// Mitsubishi GX Works2 project: GDF-UV-4GC-20210804 souce   PLC: Q00U

PROGRAM MAIN
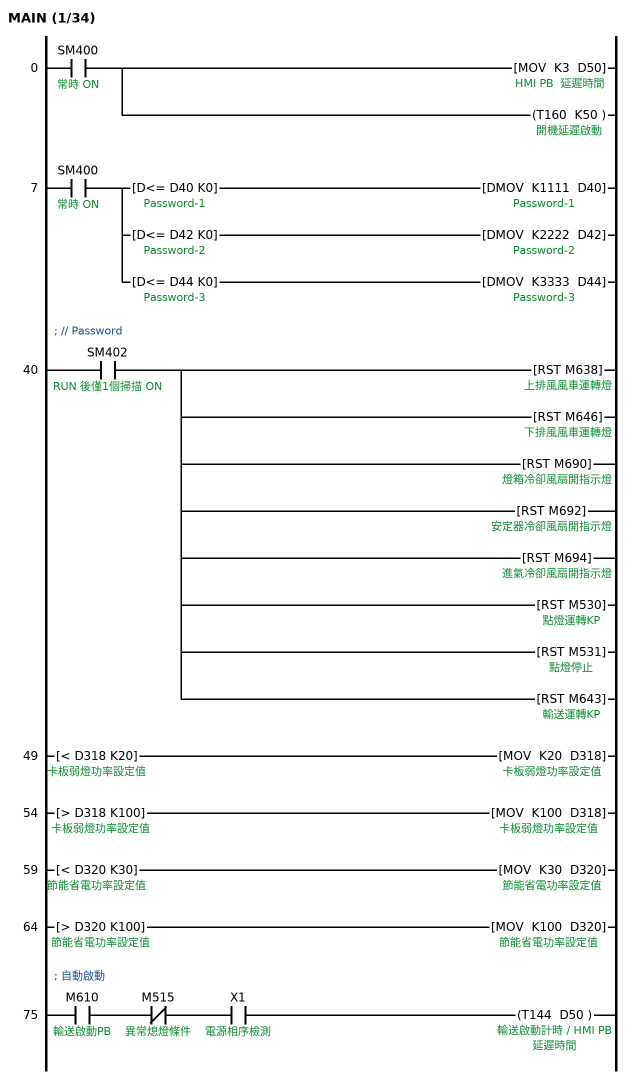
0     LD      SM400  ; 常時 ON
      MOV     K3 D50  ; HMI PB  延遲時間
      OUT     T160 K50  ; 開機延遲啟動
7     LD      SM400  ; 常時 ON
      MPS
      ANDD<=  D40 K0  ; Password-1
      DMOV    K1111 D40
      MRD
      ANDD<=  D42 K0  ; Password-2
      DMOV    K2222 D42
      MPP
      ANDD<=  D44 K0  ; Password-3
      DMOV    K3333 D44
; // Password
40    LD      SM402  ; RUN 後僅1個掃描 ON
      RST     M638  ; 上排風風車運轉燈
      RST     M646  ; 下排風風車運轉燈
      RST     M690  ; 燈箱冷卻風扇開指示燈
      RST     M692  ; 安定器冷卻風扇開指示燈
      RST     M694  ; 進氣冷卻風扇開指示燈
      RST     M530  ; 點燈運轉KP
      RST     M531  ; 點燈停止
      RST     M643  ; 輸送運轉KP
49    LD<     D318 K20  ; 卡板弱燈功率設定值
      MOV     K20 D318
54    LD>     D318 K100  ; 卡板弱燈功率設定值
      MOV     K100 D318
59    LD<     D320 K30  ; 節能省電功率設定值
      MOV     K30 D320
64    LD>     D320 K100  ; 節能省電功率設定值
      MOV     K100 D320
; 自動啟動
75    LD      M610  ; 輸送啟動PB
      ANI     M515  ; 異常熄燈條件
      AND     X1  ; 電源相序檢測
      OUT     T144 D50  ; 輸送啟動計時 / HMI PB  延遲時間
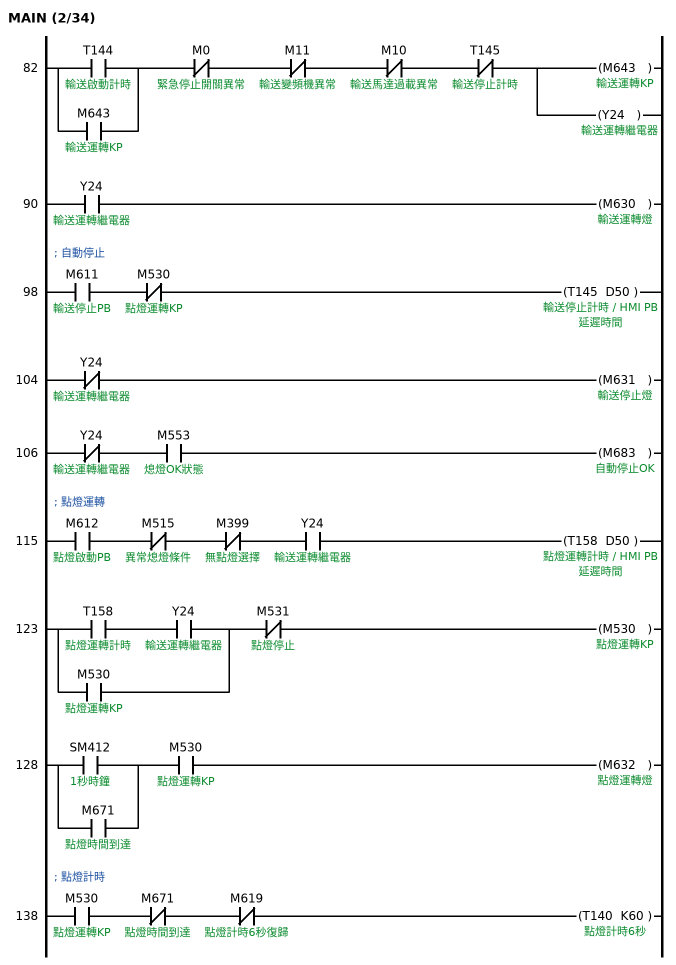
82    LD      T144  ; 輸送啟動計時
      OR      M643  ; 輸送運轉KP
      ANI     M0  ; 緊急停止開關異常
      ANI     M11  ; 輸送變頻機異常
      ANI     M10  ; 輸送馬達過載異常
      ANI     T145  ; 輸送停止計時
      OUT     M643  ; 輸送運轉KP
      OUT     Y24  ; 輸送運轉繼電器
90    LD      Y24  ; 輸送運轉繼電器
      OUT     M630  ; 輸送運轉燈
; 自動停止
98    LD      M611  ; 輸送停止PB
      ANI     M530  ; 點燈運轉KP
      OUT     T145 D50  ; 輸送停止計時 / HMI PB  延遲時間
104   LDI     Y24  ; 輸送運轉繼電器
      OUT     M631  ; 輸送停止燈
106   LDI     Y24  ; 輸送運轉繼電器
      AND     M553  ; 熄燈OK狀態
      OUT     M683  ; 自動停止OK
; 點燈運轉
115   LD      M612  ; 點燈啟動PB
      ANI     M515  ; 異常熄燈條件
      ANI     M399  ; 無點燈選擇
      AND     Y24  ; 輸送運轉繼電器
      OUT     T158 D50  ; 點燈運轉計時 / HMI PB  延遲時間
123   LD      T158  ; 點燈運轉計時
      AND     Y24  ; 輸送運轉繼電器
      OR      M530  ; 點燈運轉KP
      ANI     M531  ; 點燈停止
      OUT     M530  ; 點燈運轉KP
128   LD      SM412  ; 1秒時鐘
      OR      M671  ; 點燈時間到達
      AND     M530  ; 點燈運轉KP
      OUT     M632  ; 點燈運轉燈
; 點燈計時
138   LD      M530  ; 點燈運轉KP
      ANI     M671  ; 點燈時間到達
      ANI     M619  ; 點燈計時6秒復歸
      OUT     T140 K60  ; 點燈計時6秒
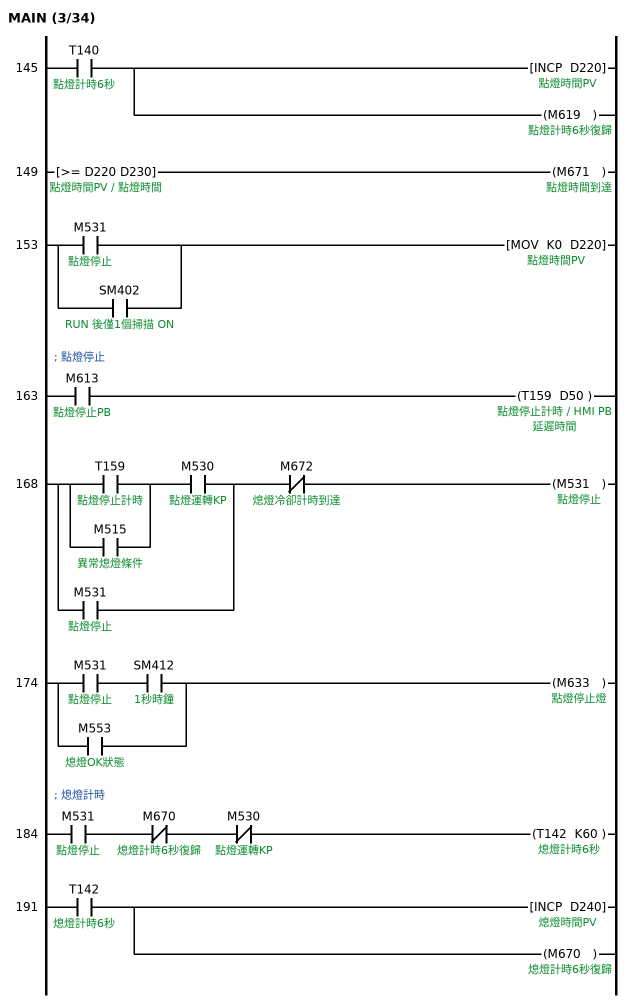
145   LD      T140  ; 點燈計時6秒
      INCP    D220  ; 點燈時間PV
      OUT     M619  ; 點燈計時6秒復歸
149   LD>=    D220 D230  ; 點燈時間PV / 點燈時間
      OUT     M671  ; 點燈時間到達
153   LD      M531  ; 點燈停止
      OR      SM402  ; RUN 後僅1個掃描 ON
      MOV     K0 D220
; 點燈停止
163   LD      M613  ; 點燈停止PB
      OUT     T159 D50  ; 點燈停止計時 / HMI PB  延遲時間
168   LD      T159  ; 點燈停止計時
      OR      M515  ; 異常熄燈條件
      AND     M530  ; 點燈運轉KP
      OR      M531  ; 點燈停止
      ANI     M672  ; 熄燈冷卻計時到達
      OUT     M531  ; 點燈停止
174   LD      M531  ; 點燈停止
      AND     SM412  ; 1秒時鐘
      OR      M553  ; 熄燈OK狀態
      OUT     M633  ; 點燈停止燈
; 熄燈計時
184   LD      M531  ; 點燈停止
      ANI     M670  ; 熄燈計時6秒復歸
      ANI     M530  ; 點燈運轉KP
      OUT     T142 K60  ; 熄燈計時6秒
191   LD      T142  ; 熄燈計時6秒
      INCP    D240  ; 熄燈時間PV
      OUT     M670  ; 熄燈計時6秒復歸
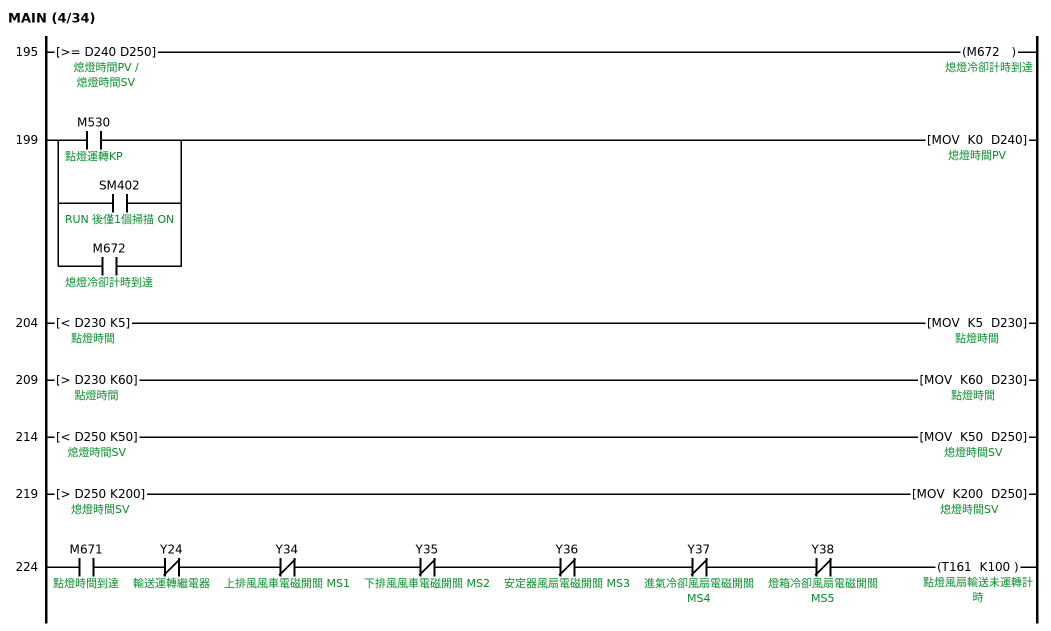
195   LD>=    D240 D250  ; 熄燈時間PV / 熄燈時間SV
      OUT     M672  ; 熄燈冷卻計時到達
199   LD      M530  ; 點燈運轉KP
      OR      SM402  ; RUN 後僅1個掃描 ON
      OR      M672  ; 熄燈冷卻計時到達
      MOV     K0 D240
204   LD<     D230 K5  ; 點燈時間
      MOV     K5 D230
209   LD>     D230 K60  ; 點燈時間
      MOV     K60 D230
214   LD<     D250 K50  ; 熄燈時間SV
      MOV     K50 D250
219   LD>     D250 K200  ; 熄燈時間SV
      MOV     K200 D250
224   LD      M671  ; 點燈時間到達
      ANI     Y24  ; 輸送運轉繼電器
      ANI     Y34  ; 上排風風車電磁開關 MS1
      ANI     Y35  ; 下排風風車電磁開關 MS2
      ANI     Y36  ; 安定器風扇電磁開關 MS3
      ANI     Y37  ; 進氣冷卻風扇電磁開關 MS4
      ANI     Y38  ; 燈箱冷卻風扇電磁開關 MS5
      OUT     T161 K100  ; 點燈風扇輸送未運轉計時
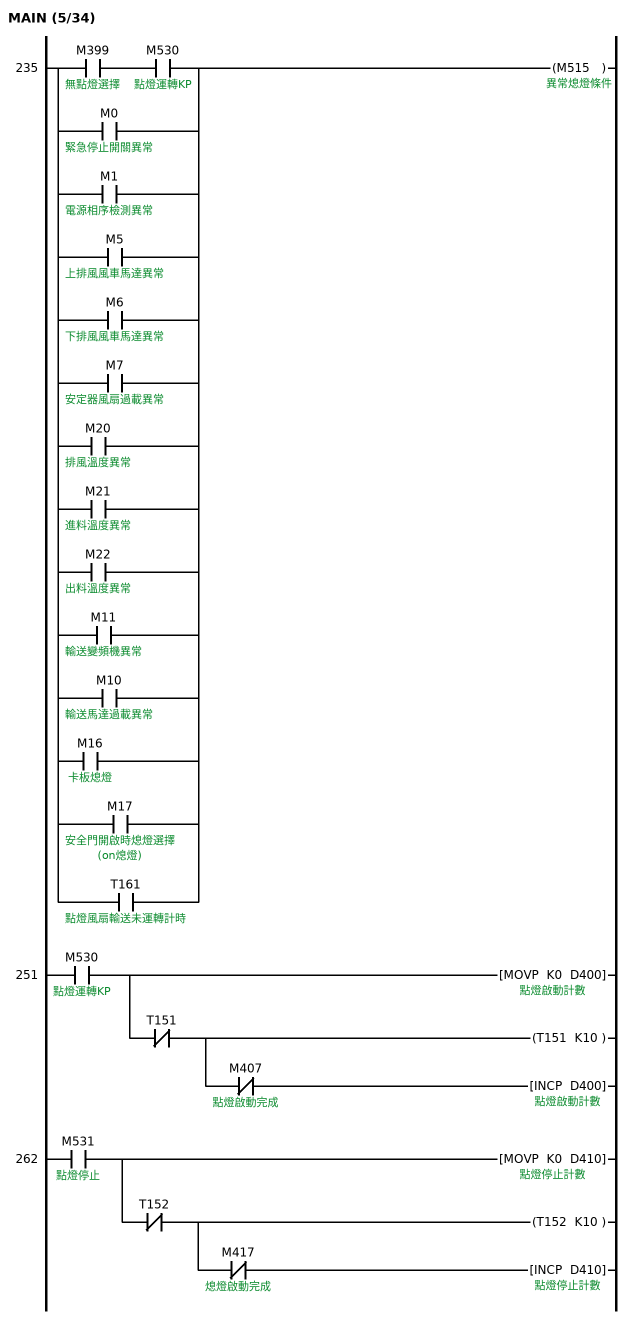
235   LD      M399  ; 無點燈選擇
      AND     M530  ; 點燈運轉KP
      OR      M0  ; 緊急停止開關異常
      OR      M1  ; 電源相序檢測異常
      OR      M5  ; 上排風風車馬達異常
      OR      M6  ; 下排風風車馬達異常
      OR      M7  ; 安定器風扇過載異常
      OR      M20  ; 排風溫度異常
      OR      M21  ; 進料溫度異常
      OR      M22  ; 出料溫度異常
      OR      M11  ; 輸送變頻機異常
      OR      M10  ; 輸送馬達過載異常
      OR      M16  ; 卡板熄燈
      OR      M17  ; 安全門開啟時熄燈選擇    (on熄燈)
      OR      T161  ; 點燈風扇輸送未運轉計時
      OUT     M515  ; 異常熄燈條件
251   LD      M530  ; 點燈運轉KP
      MOVP    K0 D400  ; 點燈啟動計數
      ANI     T151
      OUT     T151 K10
      ANI     M407  ; 點燈啟動完成
      INCP    D400
262   LD      M531  ; 點燈停止
      MOVP    K0 D410  ; 點燈停止計數
      ANI     T152
      OUT     T152 K10
      ANI     M417  ; 熄燈啟動完成
      INCP    D410
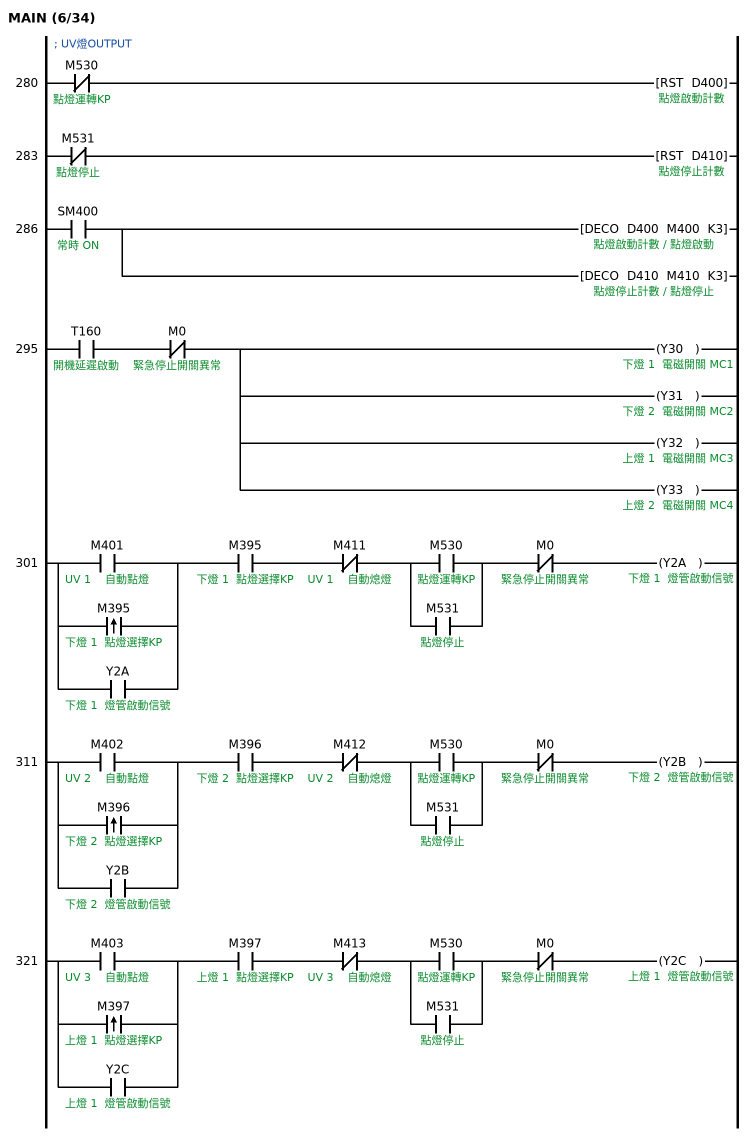
; UV燈OUTPUT
280   LDI     M530  ; 點燈運轉KP
      RST     D400  ; 點燈啟動計數
283   LDI     M531  ; 點燈停止
      RST     D410  ; 點燈停止計數
286   LD      SM400  ; 常時 ON
      DECO    D400 M400 K3  ; 點燈啟動
      DECO    D410 M410 K3  ; 點燈停止
295   LD      T160  ; 開機延遲啟動
      ANI     M0  ; 緊急停止開關異常
      OUT     Y30  ; 下燈 1  電磁開關 MC1
      OUT     Y31  ; 下燈 2  電磁開關 MC2
      OUT     Y32  ; 上燈 1  電磁開關 MC3
      OUT     Y33  ; 上燈 2  電磁開關 MC4
301   LD      M401  ; UV 1    自動點燈
      ORP     M395  ; 下燈 1  點燈選擇KP
      OR      Y2A  ; 下燈 1  燈管啟動信號
      AND     M395  ; 下燈 1  點燈選擇KP
      ANI     M411  ; UV 1    自動熄燈
      LD      M530  ; 點燈運轉KP
      OR      M531  ; 點燈停止
      ANB
      ANI     M0  ; 緊急停止開關異常
      OUT     Y2A  ; 下燈 1  燈管啟動信號
311   LD      M402  ; UV 2    自動點燈
      ORP     M396  ; 下燈 2  點燈選擇KP
      OR      Y2B  ; 下燈 2  燈管啟動信號
      AND     M396  ; 下燈 2  點燈選擇KP
      ANI     M412  ; UV 2    自動熄燈
      LD      M530  ; 點燈運轉KP
      OR      M531  ; 點燈停止
      ANB
      ANI     M0  ; 緊急停止開關異常
      OUT     Y2B  ; 下燈 2  燈管啟動信號
321   LD      M403  ; UV 3    自動點燈
      ORP     M397  ; 上燈 1  點燈選擇KP
      OR      Y2C  ; 上燈 1  燈管啟動信號
      AND     M397  ; 上燈 1  點燈選擇KP
      ANI     M413  ; UV 3    自動熄燈
      LD      M530  ; 點燈運轉KP
      OR      M531  ; 點燈停止
      ANB
      ANI     M0  ; 緊急停止開關異常
      OUT     Y2C  ; 上燈 1  燈管啟動信號
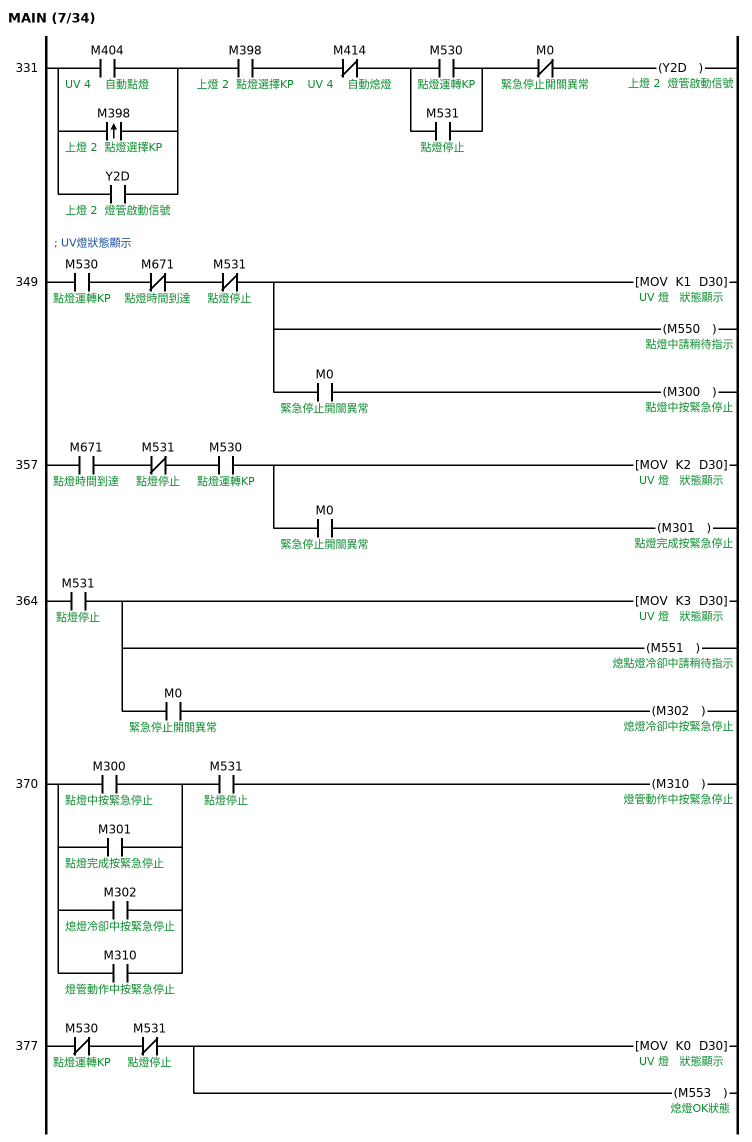
331   LD      M404  ; UV 4    自動點燈
      ORP     M398  ; 上燈 2  點燈選擇KP
      OR      Y2D  ; 上燈 2  燈管啟動信號
      AND     M398  ; 上燈 2  點燈選擇KP
      ANI     M414  ; UV 4    自動熄燈
      LD      M530  ; 點燈運轉KP
      OR      M531  ; 點燈停止
      ANB
      ANI     M0  ; 緊急停止開關異常
      OUT     Y2D  ; 上燈 2  燈管啟動信號
; UV燈狀態顯示
349   LD      M530  ; 點燈運轉KP
      ANI     M671  ; 點燈時間到達
      ANI     M531  ; 點燈停止
      MOV     K1 D30  ; UV 燈   狀態顯示
      OUT     M550  ; 點燈中請稍待指示
      AND     M0  ; 緊急停止開關異常
      OUT     M300  ; 點燈中按緊急停止
357   LD      M671  ; 點燈時間到達
      ANI     M531  ; 點燈停止
      AND     M530  ; 點燈運轉KP
      MOV     K2 D30
      AND     M0  ; 緊急停止開關異常
      OUT     M301  ; 點燈完成按緊急停止
364   LD      M531  ; 點燈停止
      MOV     K3 D30
      OUT     M551  ; 熄點燈冷卻中請稍待指示
      AND     M0  ; 緊急停止開關異常
      OUT     M302  ; 熄燈冷卻中按緊急停止
370   LD      M300  ; 點燈中按緊急停止
      OR      M301  ; 點燈完成按緊急停止
      OR      M302  ; 熄燈冷卻中按緊急停止
      OR      M310  ; 燈管動作中按緊急停止
      AND     M531  ; 點燈停止
      OUT     M310  ; 燈管動作中按緊急停止
        [note] 
377   LDI     M530  ; 點燈運轉KP
      ANI     M531  ; 點燈停止
      MOV     K0 D30
      OUT     M553  ; 熄燈OK狀態
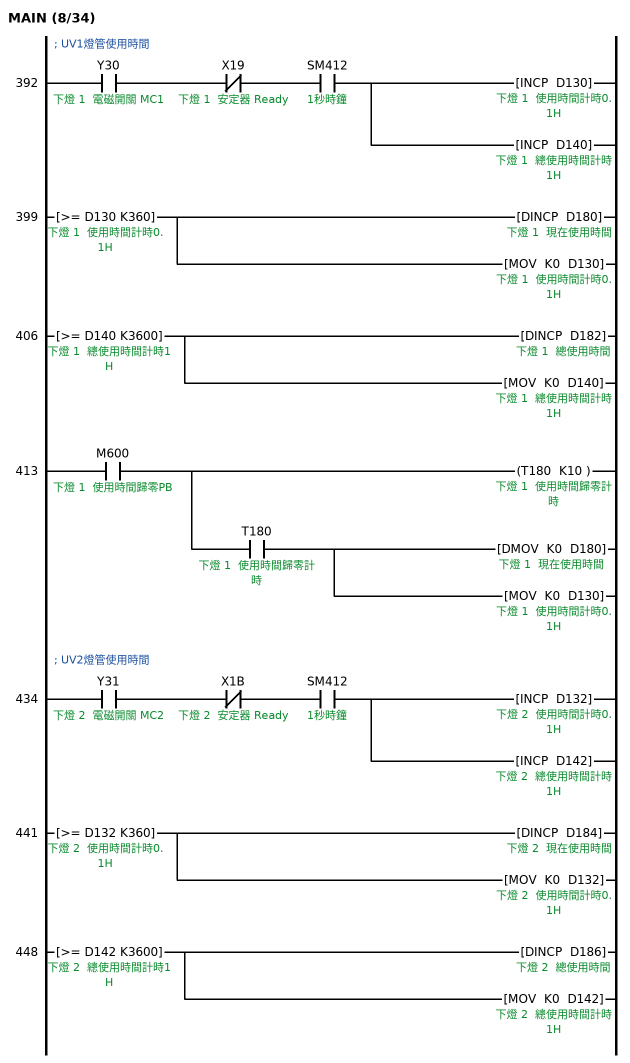
; UV1燈管使用時間
392   LD      Y30  ; 下燈 1  電磁開關 MC1
      ANI     X19  ; 下燈 1  安定器 Ready
      AND     SM412  ; 1秒時鐘
      INCP    D130  ; 下燈 1  使用時間計時0.1H
      INCP    D140  ; 下燈 1  總使用時間計時1H
399   LD>=    D130 K360  ; 下燈 1  使用時間計時0.1H
      DINCP   D180  ; 下燈 1  現在使用時間
      MOV     K0 D130
406   LD>=    D140 K3600  ; 下燈 1  總使用時間計時1H
      DINCP   D182  ; 下燈 1  總使用時間
      MOV     K0 D140
413   LD      M600  ; 下燈 1  使用時間歸零PB
      OUT     T180 K10  ; 下燈 1  使用時間歸零計時
      AND     T180  ; 下燈 1  使用時間歸零計時
      DMOV    K0 D180
      MOV     K0 D130
; UV2燈管使用時間
434   LD      Y31  ; 下燈 2  電磁開關 MC2
      ANI     X1B  ; 下燈 2  安定器 Ready
      AND     SM412  ; 1秒時鐘
      INCP    D132  ; 下燈 2  使用時間計時0.1H
      INCP    D142  ; 下燈 2  總使用時間計時1H
441   LD>=    D132 K360  ; 下燈 2  使用時間計時0.1H
      DINCP   D184  ; 下燈 2  現在使用時間
      MOV     K0 D132
448   LD>=    D142 K3600  ; 下燈 2  總使用時間計時1H
      DINCP   D186  ; 下燈 2  總使用時間
      MOV     K0 D142
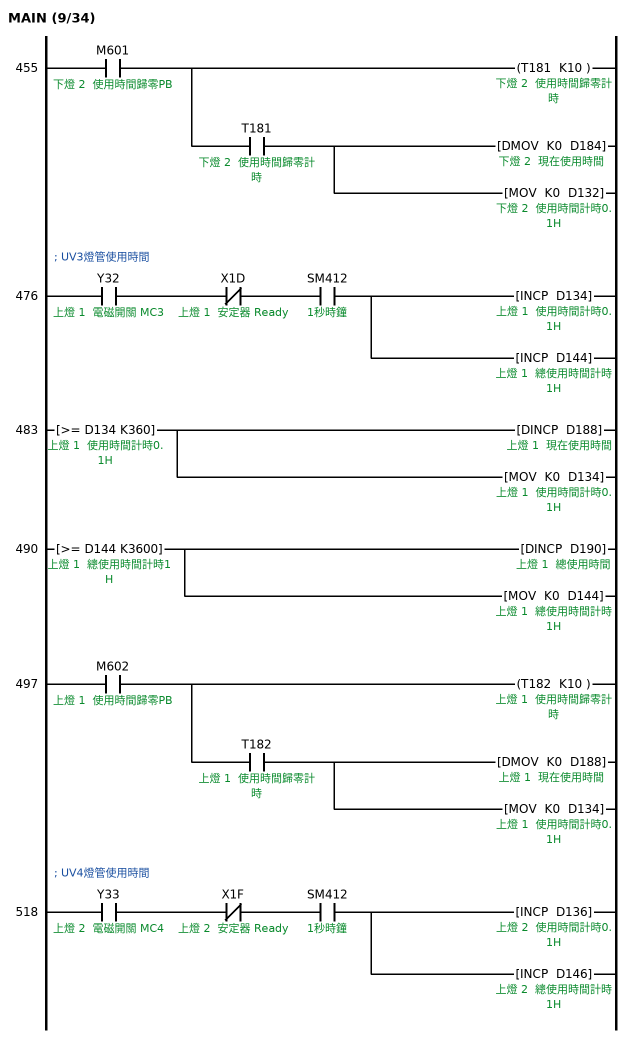
455   LD      M601  ; 下燈 2  使用時間歸零PB
      OUT     T181 K10  ; 下燈 2  使用時間歸零計時
      AND     T181  ; 下燈 2  使用時間歸零計時
      DMOV    K0 D184
      MOV     K0 D132
; UV3燈管使用時間
476   LD      Y32  ; 上燈 1  電磁開關 MC3
      ANI     X1D  ; 上燈 1  安定器 Ready
      AND     SM412  ; 1秒時鐘
      INCP    D134  ; 上燈 1  使用時間計時0.1H
      INCP    D144  ; 上燈 1  總使用時間計時1H
483   LD>=    D134 K360  ; 上燈 1  使用時間計時0.1H
      DINCP   D188  ; 上燈 1  現在使用時間
      MOV     K0 D134
490   LD>=    D144 K3600  ; 上燈 1  總使用時間計時1H
      DINCP   D190  ; 上燈 1  總使用時間
      MOV     K0 D144
497   LD      M602  ; 上燈 1  使用時間歸零PB
      OUT     T182 K10  ; 上燈 1  使用時間歸零計時
      AND     T182  ; 上燈 1  使用時間歸零計時
      DMOV    K0 D188
      MOV     K0 D134
; UV4燈管使用時間
518   LD      Y33  ; 上燈 2  電磁開關 MC4
      ANI     X1F  ; 上燈 2  安定器 Ready
      AND     SM412  ; 1秒時鐘
      INCP    D136  ; 上燈 2  使用時間計時0.1H
      INCP    D146  ; 上燈 2  總使用時間計時1H
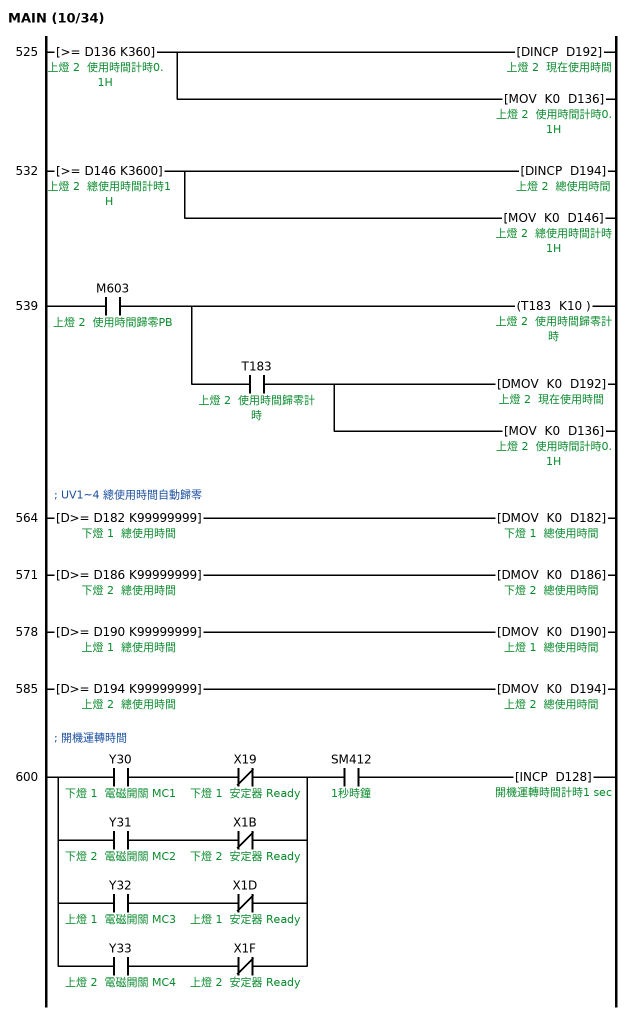
525   LD>=    D136 K360  ; 上燈 2  使用時間計時0.1H
      DINCP   D192  ; 上燈 2  現在使用時間
      MOV     K0 D136
532   LD>=    D146 K3600  ; 上燈 2  總使用時間計時1H
      DINCP   D194  ; 上燈 2  總使用時間
      MOV     K0 D146
539   LD      M603  ; 上燈 2  使用時間歸零PB
      OUT     T183 K10  ; 上燈 2  使用時間歸零計時
      AND     T183  ; 上燈 2  使用時間歸零計時
      DMOV    K0 D192
      MOV     K0 D136
; UV1~4 總使用時間自動歸零
564   LDD>=   D182 K99999999  ; 下燈 1  總使用時間
      DMOV    K0 D182
571   LDD>=   D186 K99999999  ; 下燈 2  總使用時間
      DMOV    K0 D186
578   LDD>=   D190 K99999999  ; 上燈 1  總使用時間
      DMOV    K0 D190
585   LDD>=   D194 K99999999  ; 上燈 2  總使用時間
      DMOV    K0 D194
; 開機運轉時間
600   LD      Y30  ; 下燈 1  電磁開關 MC1
      ANI     X19  ; 下燈 1  安定器 Ready
      LD      Y31  ; 下燈 2  電磁開關 MC2
      ANI     X1B  ; 下燈 2  安定器 Ready
      ORB
      LD      Y32  ; 上燈 1  電磁開關 MC3
      ANI     X1D  ; 上燈 1  安定器 Ready
      ORB
      LD      Y33  ; 上燈 2  電磁開關 MC4
      ANI     X1F  ; 上燈 2  安定器 Ready
      ORB
      AND     SM412  ; 1秒時鐘
      INCP    D128  ; 開機運轉時間計時1 sec
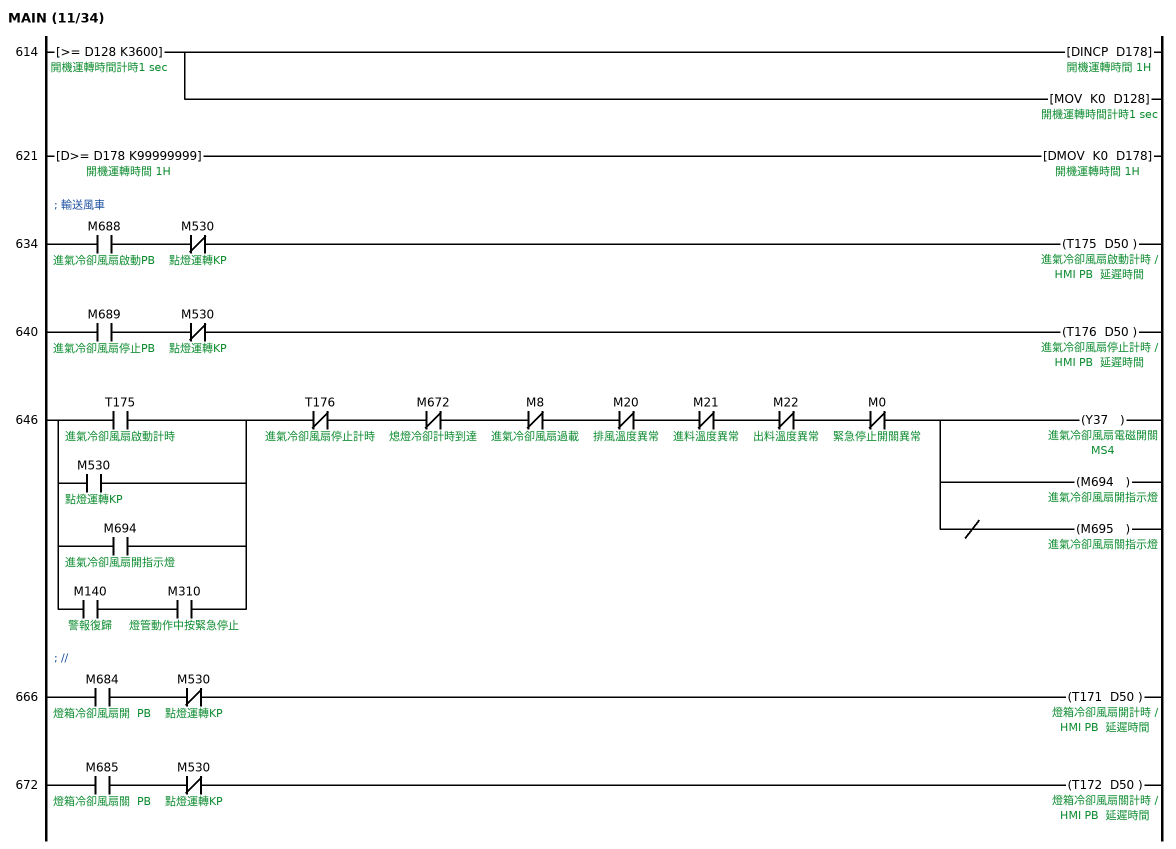
614   LD>=    D128 K3600  ; 開機運轉時間計時1 sec
      DINCP   D178  ; 開機運轉時間 1H
      MOV     K0 D128
621   LDD>=   D178 K99999999  ; 開機運轉時間 1H
      DMOV    K0 D178
; 輸送風車
634   LD      M688  ; 進氣冷卻風扇啟動PB
      ANI     M530  ; 點燈運轉KP
      OUT     T175 D50  ; 進氣冷卻風扇啟動計時 / HMI PB  延遲時間
640   LD      M689  ; 進氣冷卻風扇停止PB
      ANI     M530  ; 點燈運轉KP
      OUT     T176 D50  ; 進氣冷卻風扇停止計時 / HMI PB  延遲時間
646   LD      T175  ; 進氣冷卻風扇啟動計時
      OR      M530  ; 點燈運轉KP
      OR      M694  ; 進氣冷卻風扇開指示燈
      LD      M140  ; 警報復歸
      AND     M310  ; 燈管動作中按緊急停止
      ORB
      ANI     T176  ; 進氣冷卻風扇停止計時
      ANI     M672  ; 熄燈冷卻計時到達
      ANI     M8  ; 進氣冷卻風扇過載
      ANI     M20  ; 排風溫度異常
      ANI     M21  ; 進料溫度異常
      ANI     M22  ; 出料溫度異常
      ANI     M0  ; 緊急停止開關異常
      OUT     Y37  ; 進氣冷卻風扇電磁開關 MS4
      OUT     M694  ; 進氣冷卻風扇開指示燈
      INV
      OUT     M695  ; 進氣冷卻風扇關指示燈
; //
666   LD      M684  ; 燈箱冷卻風扇開  PB
      ANI     M530  ; 點燈運轉KP
      OUT     T171 D50  ; 燈箱冷卻風扇開計時 / HMI PB  延遲時間
672   LD      M685  ; 燈箱冷卻風扇關  PB
      ANI     M530  ; 點燈運轉KP
      OUT     T172 D50  ; 燈箱冷卻風扇關計時 / HMI PB  延遲時間
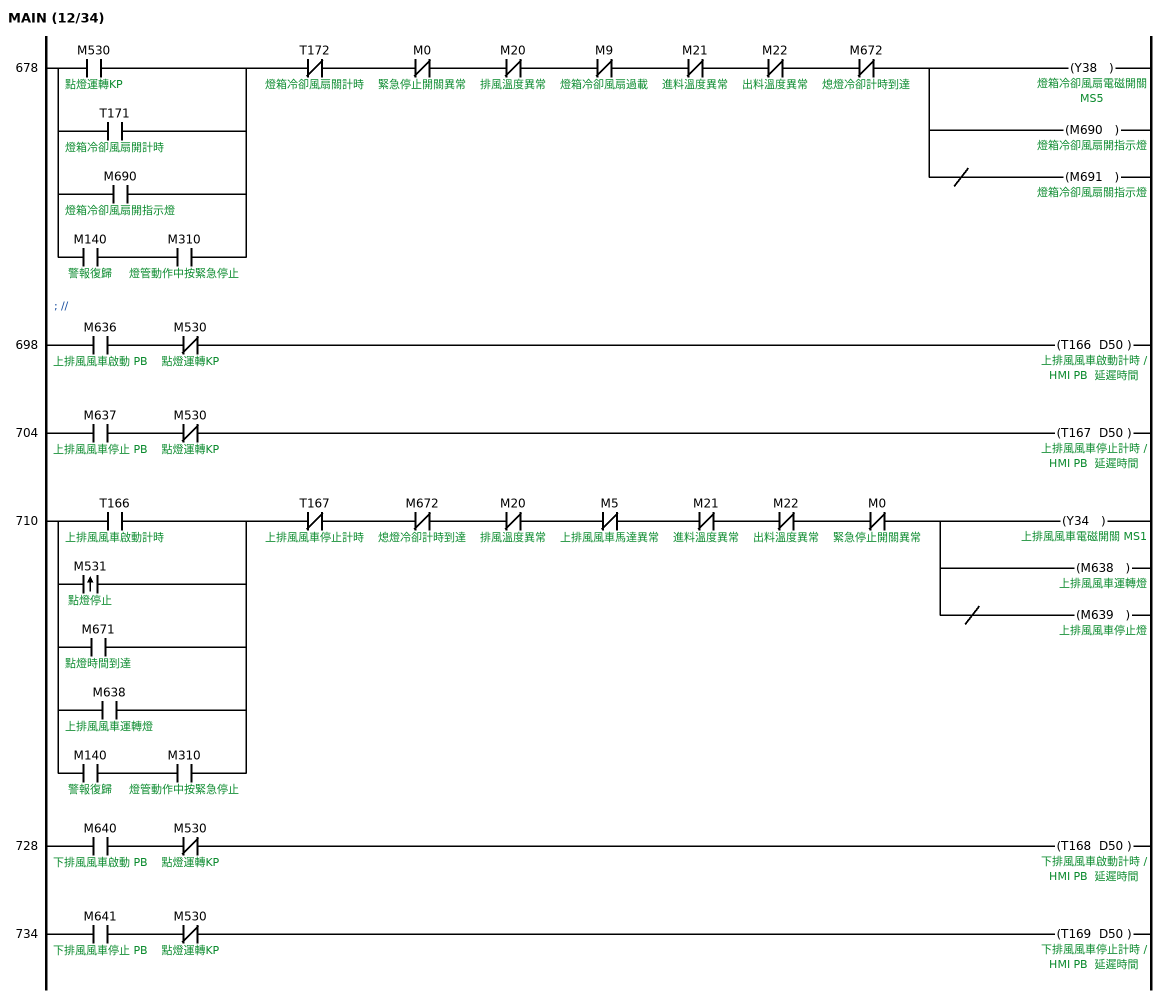
678   LD      M530  ; 點燈運轉KP
      OR      T171  ; 燈箱冷卻風扇開計時
      OR      M690  ; 燈箱冷卻風扇開指示燈
      LD      M140  ; 警報復歸
      AND     M310  ; 燈管動作中按緊急停止
      ORB
      ANI     T172  ; 燈箱冷卻風扇關計時
      ANI     M0  ; 緊急停止開關異常
      ANI     M20  ; 排風溫度異常
      ANI     M9  ; 燈箱冷卻風扇過載
      ANI     M21  ; 進料溫度異常
      ANI     M22  ; 出料溫度異常
      ANI     M672  ; 熄燈冷卻計時到達
      OUT     Y38  ; 燈箱冷卻風扇電磁開關 MS5
      OUT     M690  ; 燈箱冷卻風扇開指示燈
      INV
      OUT     M691  ; 燈箱冷卻風扇關指示燈
; //
698   LD      M636  ; 上排風風車啟動 PB
      ANI     M530  ; 點燈運轉KP
      OUT     T166 D50  ; 上排風風車啟動計時 / HMI PB  延遲時間
704   LD      M637  ; 上排風風車停止 PB
      ANI     M530  ; 點燈運轉KP
      OUT     T167 D50  ; 上排風風車停止計時 / HMI PB  延遲時間
710   LD      T166  ; 上排風風車啟動計時
      ORP     M531  ; 點燈停止
      OR      M671  ; 點燈時間到達
      OR      M638  ; 上排風風車運轉燈
      LD      M140  ; 警報復歸
      AND     M310  ; 燈管動作中按緊急停止
      ORB
      ANI     T167  ; 上排風風車停止計時
      ANI     M672  ; 熄燈冷卻計時到達
      ANI     M20  ; 排風溫度異常
      ANI     M5  ; 上排風風車馬達異常
      ANI     M21  ; 進料溫度異常
      ANI     M22  ; 出料溫度異常
      ANI     M0  ; 緊急停止開關異常
      OUT     Y34  ; 上排風風車電磁開關 MS1
      OUT     M638  ; 上排風風車運轉燈
      INV
      OUT     M639  ; 上排風風車停止燈
728   LD      M640  ; 下排風風車啟動 PB
      ANI     M530  ; 點燈運轉KP
      OUT     T168 D50  ; 下排風風車啟動計時 / HMI PB  延遲時間
734   LD      M641  ; 下排風風車停止 PB
      ANI     M530  ; 點燈運轉KP
      OUT     T169 D50  ; 下排風風車停止計時 / HMI PB  延遲時間
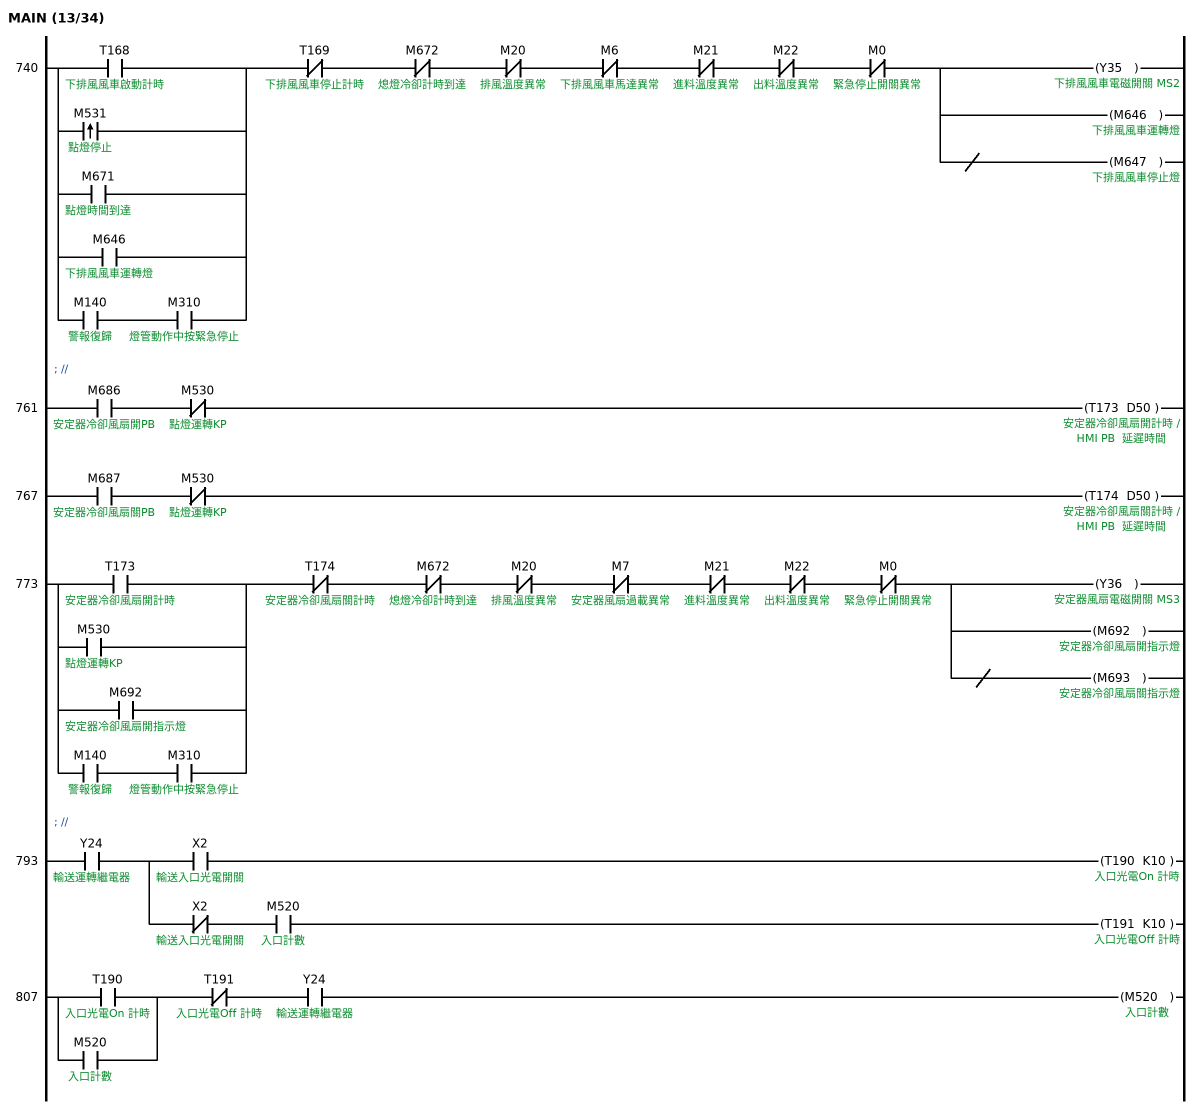
740   LD      T168  ; 下排風風車啟動計時
      ORP     M531  ; 點燈停止
      OR      M671  ; 點燈時間到達
      OR      M646  ; 下排風風車運轉燈
      LD      M140  ; 警報復歸
      AND     M310  ; 燈管動作中按緊急停止
      ORB
      ANI     T169  ; 下排風風車停止計時
      ANI     M672  ; 熄燈冷卻計時到達
      ANI     M20  ; 排風溫度異常
      ANI     M6  ; 下排風風車馬達異常
      ANI     M21  ; 進料溫度異常
      ANI     M22  ; 出料溫度異常
      ANI     M0  ; 緊急停止開關異常
      OUT     Y35  ; 下排風風車電磁開關 MS2
      OUT     M646  ; 下排風風車運轉燈
      INV
      OUT     M647  ; 下排風風車停止燈
; //
761   LD      M686  ; 安定器冷卻風扇開PB
      ANI     M530  ; 點燈運轉KP
      OUT     T173 D50  ; 安定器冷卻風扇開計時 / HMI PB  延遲時間
767   LD      M687  ; 安定器冷卻風扇關PB
      ANI     M530  ; 點燈運轉KP
      OUT     T174 D50  ; 安定器冷卻風扇關計時 / HMI PB  延遲時間
773   LD      T173  ; 安定器冷卻風扇開計時
      OR      M530  ; 點燈運轉KP
      OR      M692  ; 安定器冷卻風扇開指示燈
      LD      M140  ; 警報復歸
      AND     M310  ; 燈管動作中按緊急停止
      ORB
      ANI     T174  ; 安定器冷卻風扇關計時
      ANI     M672  ; 熄燈冷卻計時到達
      ANI     M20  ; 排風溫度異常
      ANI     M7  ; 安定器風扇過載異常
      ANI     M21  ; 進料溫度異常
      ANI     M22  ; 出料溫度異常
      ANI     M0  ; 緊急停止開關異常
      OUT     Y36  ; 安定器風扇電磁開關 MS3
      OUT     M692  ; 安定器冷卻風扇開指示燈
      INV
      OUT     M693  ; 安定器冷卻風扇關指示燈
; //
793   LD      Y24  ; 輸送運轉繼電器
      MPS
      AND     X2  ; 輸送入口光電開關
      OUT     T190 K10  ; 入口光電On 計時
      MPP
      ANI     X2  ; 輸送入口光電開關
      AND     M520  ; 入口計數
      OUT     T191 K10  ; 入口光電Off 計時
807   LD      T190  ; 入口光電On 計時
      OR      M520  ; 入口計數
      ANI     T191  ; 入口光電Off 計時
      AND     Y24  ; 輸送運轉繼電器
      OUT     M520  ; 入口計數
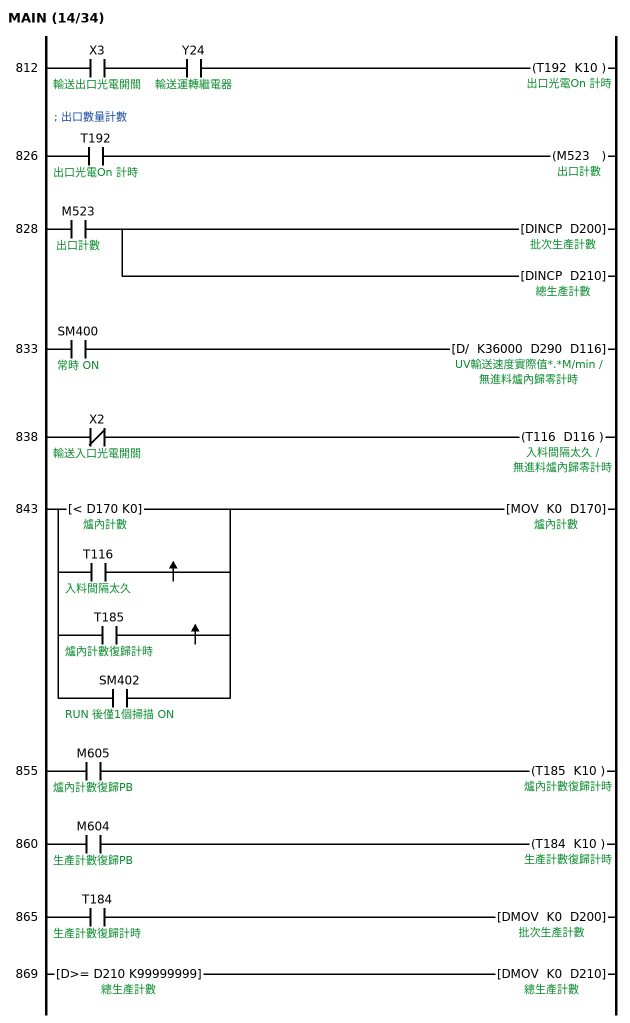
812   LD      X3  ; 輸送出口光電開關
      AND     Y24  ; 輸送運轉繼電器
      OUT     T192 K10  ; 出口光電On 計時
; 出口數量計數
826   LD      T192  ; 出口光電On 計時
      OUT     M523  ; 出口計數
828   LD      M523  ; 出口計數
      DINCP   D200  ; 批次生產計數
      DINCP   D210  ; 總生產計數
833   LD      SM400  ; 常時 ON
      D/      K36000 D290 D116  ; UV輸送速度實際值*.*M/min / 無進料爐內歸零計時
838   LDI     X2  ; 輸送入口光電開關
      OUT     T116 D116  ; 入料間隔太久 / 無進料爐內歸零計時
843   LD<     D170 K0  ; 爐內計數
      LD      T116  ; 入料間隔太久
      MEP
      ORB
      LD      T185  ; 爐內計數復歸計時
      MEP
      ORB
      OR      SM402  ; RUN 後僅1個掃描 ON
      MOV     K0 D170
855   LD      M605  ; 爐內計數復歸PB
      OUT     T185 K10  ; 爐內計數復歸計時
860   LD      M604  ; 生產計數復歸PB
      OUT     T184 K10  ; 生產計數復歸計時
865   LD      T184  ; 生產計數復歸計時
      DMOV    K0 D200
869   LDD>=   D210 K99999999  ; 總生產計數
      DMOV    K0 D210
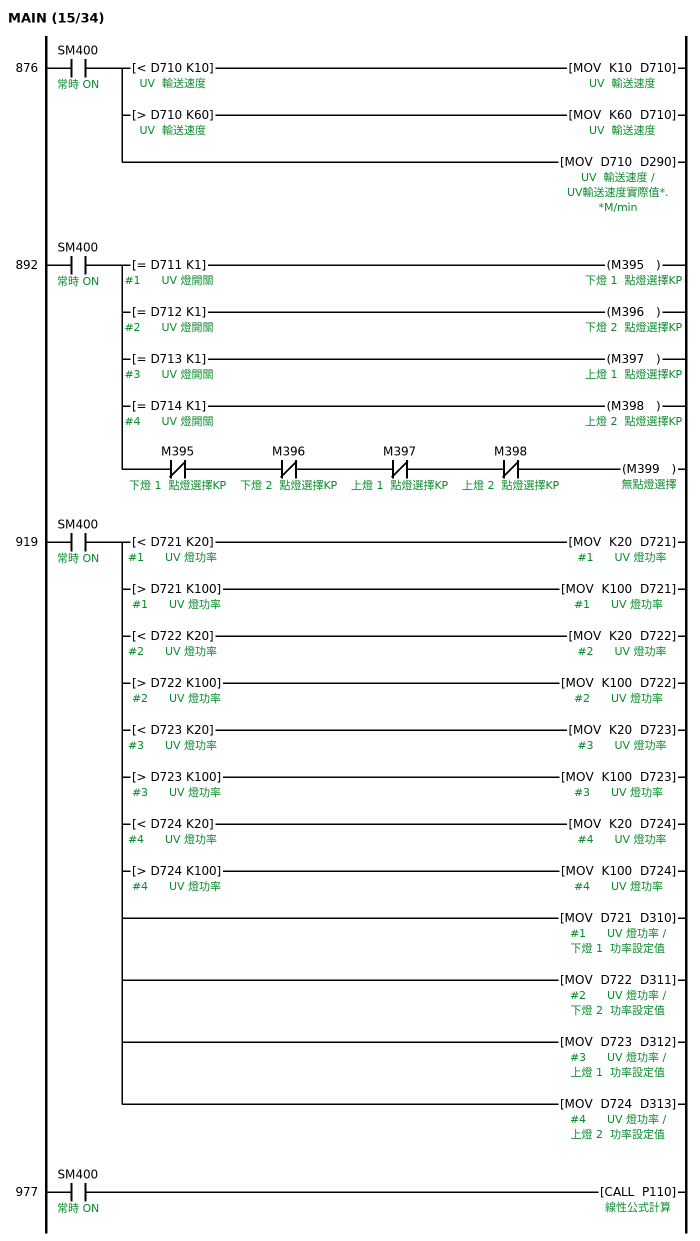
876   LD      SM400  ; 常時 ON
      MPS
      AND<    D710 K10  ; UV  輸送速度
      MOV     K10 D710
      MRD
      AND>    D710 K60  ; UV  輸送速度
      MOV     K60 D710
      MPP
      MOV     D710 D290
892   LD      SM400  ; 常時 ON
      MPS
      AND=    D711 K1  ; #1      UV 燈開關
      OUT     M395  ; 下燈 1  點燈選擇KP
      MRD
      AND=    D712 K1  ; #2      UV 燈開關
      OUT     M396  ; 下燈 2  點燈選擇KP
      MRD
      AND=    D713 K1  ; #3      UV 燈開關
      OUT     M397  ; 上燈 1  點燈選擇KP
      MRD
      AND=    D714 K1  ; #4      UV 燈開關
      OUT     M398  ; 上燈 2  點燈選擇KP
      MPP
      ANI     M395  ; 下燈 1  點燈選擇KP
      ANI     M396  ; 下燈 2  點燈選擇KP
      ANI     M397  ; 上燈 1  點燈選擇KP
      ANI     M398  ; 上燈 2  點燈選擇KP
      OUT     M399  ; 無點燈選擇
919   LD      SM400  ; 常時 ON
      MPS
      AND<    D721 K20  ; #1      UV 燈功率
      MOV     K20 D721
      MRD
      AND>    D721 K100  ; #1      UV 燈功率
      MOV     K100 D721
      MRD
      AND<    D722 K20  ; #2      UV 燈功率
      MOV     K20 D722
      MRD
      AND>    D722 K100  ; #2      UV 燈功率
      MOV     K100 D722
      MRD
      AND<    D723 K20  ; #3      UV 燈功率
      MOV     K20 D723
      MRD
      AND>    D723 K100  ; #3      UV 燈功率
      MOV     K100 D723
      MRD
      AND<    D724 K20  ; #4      UV 燈功率
      MOV     K20 D724
      MRD
      AND>    D724 K100  ; #4      UV 燈功率
      MOV     K100 D724
      MPP
      MOV     D721 D310  ; 下燈 1  功率設定值
      MOV     D722 D311  ; 下燈 2  功率設定值
      MOV     D723 D312  ; 上燈 1  功率設定值
      MOV     D724 D313  ; 上燈 2  功率設定值
977   LD      SM400  ; 常時 ON
      CALL    P110  ; 線性公式計算
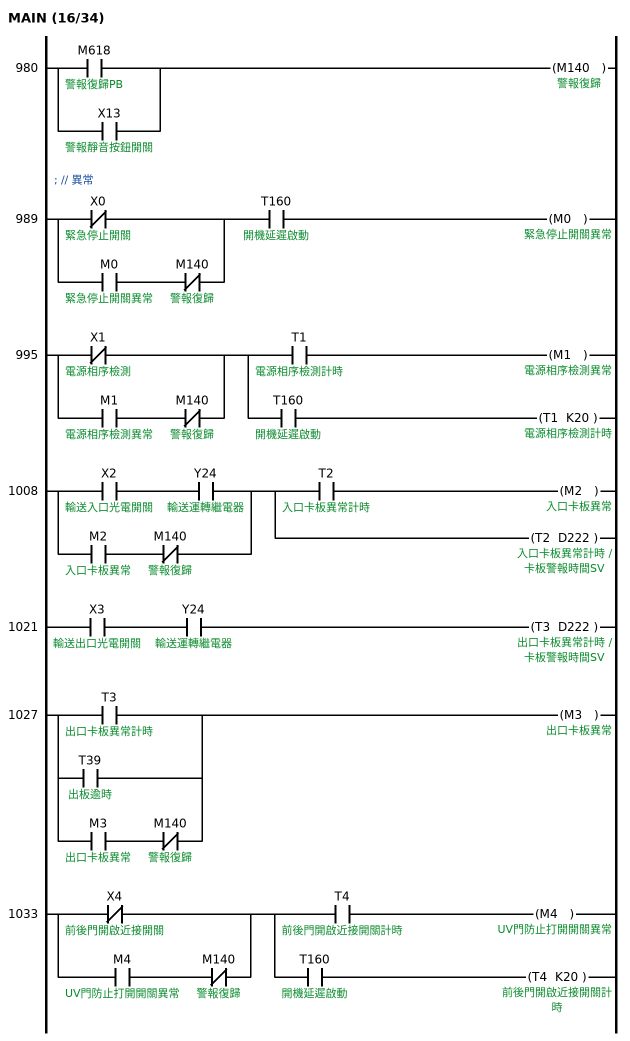
980   LD      M618  ; 警報復歸PB
      OR      X13  ; 警報靜音按鈕開關
      OUT     M140  ; 警報復歸
; // 異常
989   LDI     X0  ; 緊急停止開關
      LD      M0  ; 緊急停止開關異常
      ANI     M140  ; 警報復歸
      ORB
      AND     T160  ; 開機延遲啟動
      OUT     M0  ; 緊急停止開關異常
995   LDI     X1  ; 電源相序檢測
      LD      M1  ; 電源相序檢測異常
      ANI     M140  ; 警報復歸
      ORB
      MPS
      AND     T1  ; 電源相序檢測計時
      OUT     M1  ; 電源相序檢測異常
      MPP
      AND     T160  ; 開機延遲啟動
      OUT     T1 K20  ; 電源相序檢測計時
1008  LD      X2  ; 輸送入口光電開關
      AND     Y24  ; 輸送運轉繼電器
      LD      M2  ; 入口卡板異常
      ANI     M140  ; 警報復歸
      ORB
      MPS
      AND     T2  ; 入口卡板異常計時
      OUT     M2  ; 入口卡板異常
      MPP
      OUT     T2 D222  ; 入口卡板異常計時 / 卡板警報時間SV
1021  LD      X3  ; 輸送出口光電開關
      AND     Y24  ; 輸送運轉繼電器
      OUT     T3 D222  ; 出口卡板異常計時 / 卡板警報時間SV
1027  LD      T3  ; 出口卡板異常計時
      OR      T39  ; 出板逾時
      LD      M3  ; 出口卡板異常
      ANI     M140  ; 警報復歸
      ORB
      OUT     M3  ; 出口卡板異常
1033  LDI     X4  ; 前後門開啟近接開關
      LD      M4  ; UV門防止打開開關異常
      ANI     M140  ; 警報復歸
      ORB
      MPS
      AND     T4  ; 前後門開啟近接開關計時
      OUT     M4  ; UV門防止打開開關異常
      MPP
      AND     T160  ; 開機延遲啟動
      OUT     T4 K20  ; 前後門開啟近接開關計時
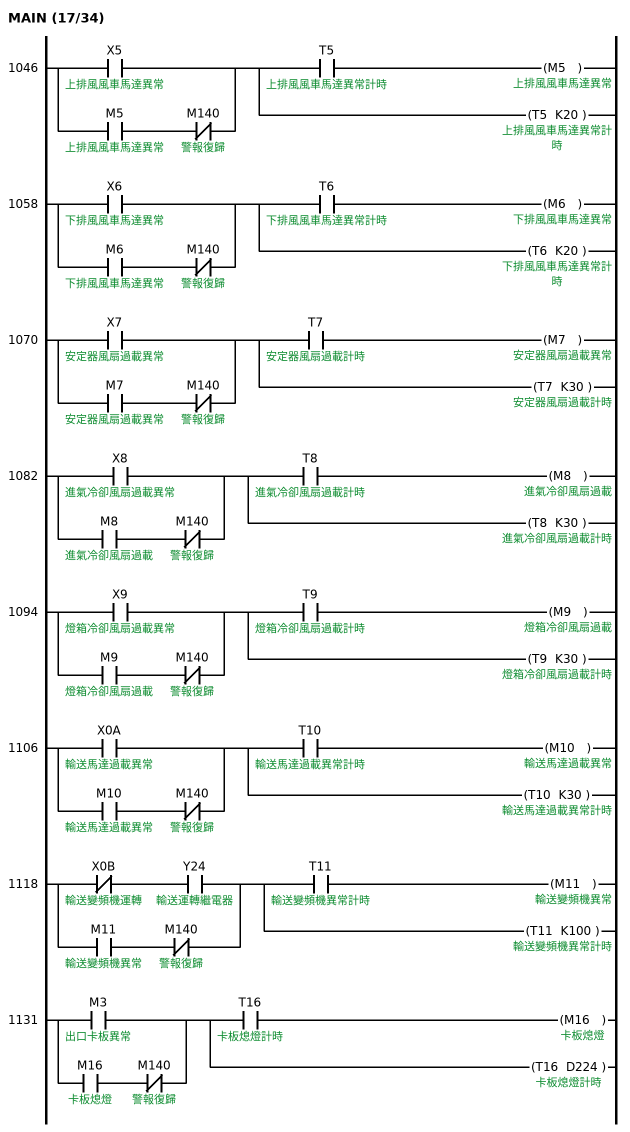
1046  LD      X5  ; 上排風風車馬達異常
      LD      M5  ; 上排風風車馬達異常
      ANI     M140  ; 警報復歸
      ORB
      MPS
      AND     T5  ; 上排風風車馬達異常計時
      OUT     M5  ; 上排風風車馬達異常
      MPP
      OUT     T5 K20  ; 上排風風車馬達異常計時
1058  LD      X6  ; 下排風風車馬達異常
      LD      M6  ; 下排風風車馬達異常
      ANI     M140  ; 警報復歸
      ORB
      MPS
      AND     T6  ; 下排風風車馬達異常計時
      OUT     M6  ; 下排風風車馬達異常
      MPP
      OUT     T6 K20  ; 下排風風車馬達異常計時
1070  LD      X7  ; 安定器風扇過載異常
      LD      M7  ; 安定器風扇過載異常
      ANI     M140  ; 警報復歸
      ORB
      MPS
      AND     T7  ; 安定器風扇過載計時
      OUT     M7  ; 安定器風扇過載異常
      MPP
      OUT     T7 K30  ; 安定器風扇過載計時
1082  LD      X8  ; 進氣冷卻風扇過載異常
      LD      M8  ; 進氣冷卻風扇過載
      ANI     M140  ; 警報復歸
      ORB
      MPS
      AND     T8  ; 進氣冷卻風扇過載計時
      OUT     M8  ; 進氣冷卻風扇過載
      MPP
      OUT     T8 K30  ; 進氣冷卻風扇過載計時
1094  LD      X9  ; 燈箱冷卻風扇過載異常
      LD      M9  ; 燈箱冷卻風扇過載
      ANI     M140  ; 警報復歸
      ORB
      MPS
      AND     T9  ; 燈箱冷卻風扇過載計時
      OUT     M9  ; 燈箱冷卻風扇過載
      MPP
      OUT     T9 K30  ; 燈箱冷卻風扇過載計時
1106  LD      X0A  ; 輸送馬達過載異常
      LD      M10  ; 輸送馬達過載異常
      ANI     M140  ; 警報復歸
      ORB
      MPS
      AND     T10  ; 輸送馬達過載異常計時
      OUT     M10  ; 輸送馬達過載異常
      MPP
      OUT     T10 K30  ; 輸送馬達過載異常計時
1118  LDI     X0B  ; 輸送變頻機運轉
      AND     Y24  ; 輸送運轉繼電器
      LD      M11  ; 輸送變頻機異常
      ANI     M140  ; 警報復歸
      ORB
      MPS
      AND     T11  ; 輸送變頻機異常計時
      OUT     M11  ; 輸送變頻機異常
      MPP
      OUT     T11 K100  ; 輸送變頻機異常計時
1131  LD      M3  ; 出口卡板異常
      LD      M16  ; 卡板熄燈
      ANI     M140  ; 警報復歸
      ORB
      MPS
      AND     T16  ; 卡板熄燈計時
      OUT     M16  ; 卡板熄燈
      MPP
      OUT     T16 D224  ; 卡板熄燈計時
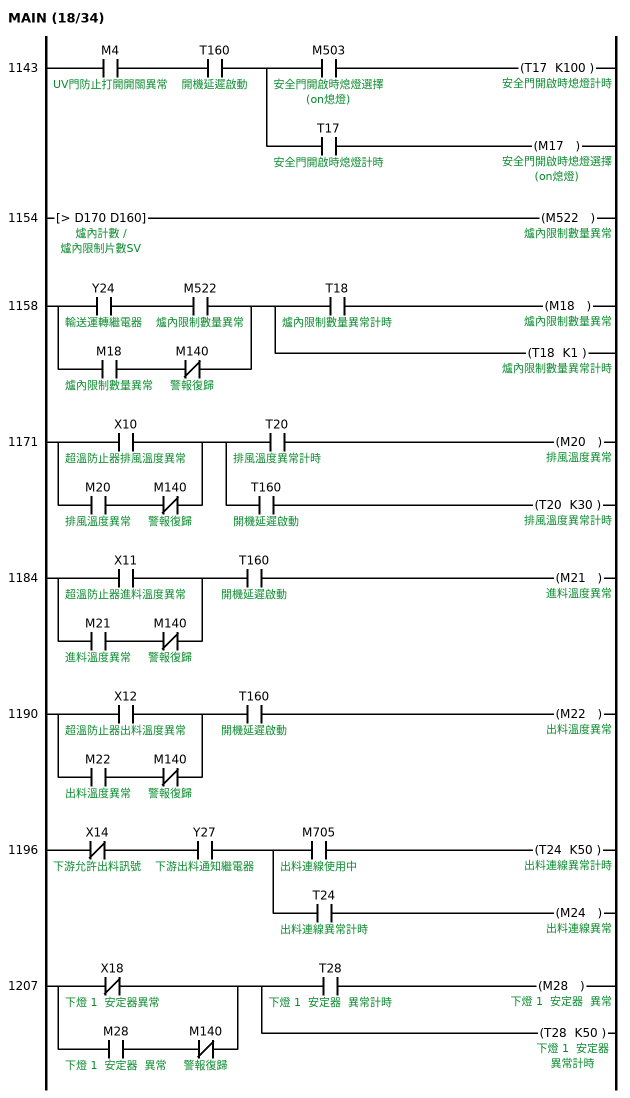
1143  LD      M4  ; UV門防止打開開關異常
      AND     T160  ; 開機延遲啟動
      MPS
      AND     M503  ; 安全門開啟時熄燈選擇    (on熄燈)
      OUT     T17 K100  ; 安全門開啟時熄燈計時
      MPP
      AND     T17  ; 安全門開啟時熄燈計時
      OUT     M17  ; 安全門開啟時熄燈選擇    (on熄燈)
1154  LD>     D170 D160  ; 爐內計數 / 爐內限制片數SV
      OUT     M522  ; 爐內限制數量異常
1158  LD      Y24  ; 輸送運轉繼電器
      AND     M522  ; 爐內限制數量異常
      LD      M18  ; 爐內限制數量異常
      ANI     M140  ; 警報復歸
      ORB
      MPS
      AND     T18  ; 爐內限制數量異常計時
      OUT     M18  ; 爐內限制數量異常
      MPP
      OUT     T18 K1  ; 爐內限制數量異常計時
1171  LD      X10  ; 超溫防止器排風溫度異常
      LD      M20  ; 排風溫度異常
      ANI     M140  ; 警報復歸
      ORB
      MPS
      AND     T20  ; 排風溫度異常計時
      OUT     M20  ; 排風溫度異常
      MPP
      AND     T160  ; 開機延遲啟動
      OUT     T20 K30  ; 排風溫度異常計時
1184  LD      X11  ; 超溫防止器進料溫度異常
      LD      M21  ; 進料溫度異常
      ANI     M140  ; 警報復歸
      ORB
      AND     T160  ; 開機延遲啟動
      OUT     M21  ; 進料溫度異常
1190  LD      X12  ; 超溫防止器出料溫度異常
      LD      M22  ; 出料溫度異常
      ANI     M140  ; 警報復歸
      ORB
      AND     T160  ; 開機延遲啟動
      OUT     M22  ; 出料溫度異常
1196  LDI     X14  ; 下游允許出料訊號
      AND     Y27  ; 下游出料通知繼電器
      MPS
      AND     M705  ; 出料連線使用中
      OUT     T24 K50  ; 出料連線異常計時
      MPP
      AND     T24  ; 出料連線異常計時
      OUT     M24  ; 出料連線異常
1207  LDI     X18  ; 下燈 1  安定器異常
      LD      M28  ; 下燈 1  安定器  異常
      ANI     M140  ; 警報復歸
      ORB
      MPS
      AND     T28  ; 下燈 1  安定器  異常計時
      OUT     M28  ; 下燈 1  安定器  異常
      MPP
      OUT     T28 K50  ; 下燈 1  安定器  異常計時
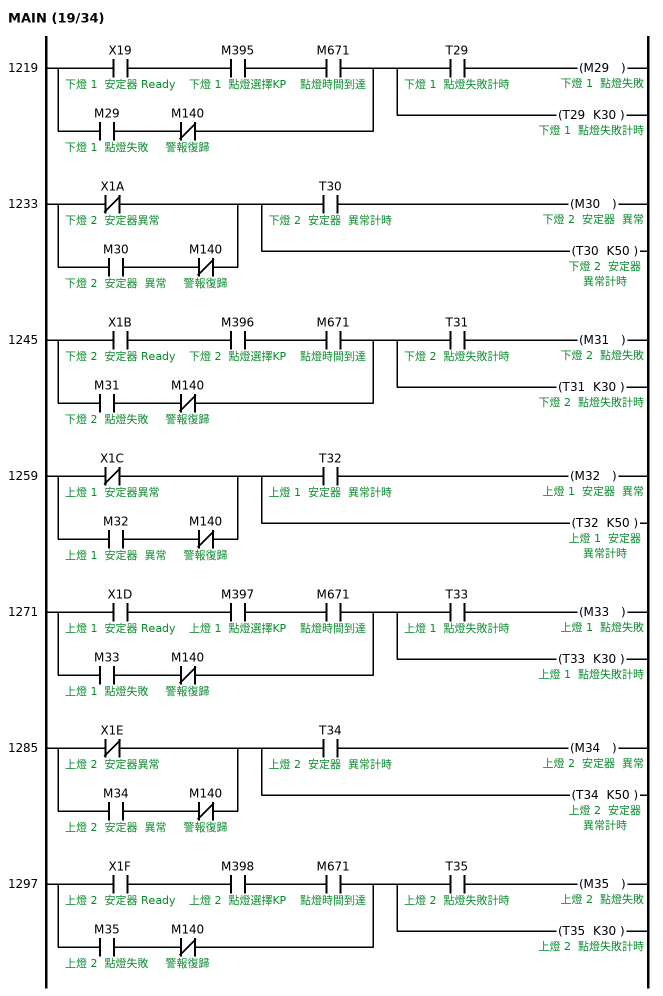
1219  LD      X19  ; 下燈 1  安定器 Ready
      AND     M395  ; 下燈 1  點燈選擇KP
      AND     M671  ; 點燈時間到達
      LD      M29  ; 下燈 1  點燈失敗
      ANI     M140  ; 警報復歸
      ORB
      MPS
      AND     T29  ; 下燈 1  點燈失敗計時
      OUT     M29  ; 下燈 1  點燈失敗
      MPP
      OUT     T29 K30  ; 下燈 1  點燈失敗計時
1233  LDI     X1A  ; 下燈 2  安定器異常
      LD      M30  ; 下燈 2  安定器  異常
      ANI     M140  ; 警報復歸
      ORB
      MPS
      AND     T30  ; 下燈 2  安定器  異常計時
      OUT     M30  ; 下燈 2  安定器  異常
      MPP
      OUT     T30 K50  ; 下燈 2  安定器  異常計時
1245  LD      X1B  ; 下燈 2  安定器 Ready
      AND     M396  ; 下燈 2  點燈選擇KP
      AND     M671  ; 點燈時間到達
      LD      M31  ; 下燈 2  點燈失敗
      ANI     M140  ; 警報復歸
      ORB
      MPS
      AND     T31  ; 下燈 2  點燈失敗計時
      OUT     M31  ; 下燈 2  點燈失敗
      MPP
      OUT     T31 K30  ; 下燈 2  點燈失敗計時
1259  LDI     X1C  ; 上燈 1  安定器異常
      LD      M32  ; 上燈 1  安定器  異常
      ANI     M140  ; 警報復歸
      ORB
      MPS
      AND     T32  ; 上燈 1  安定器  異常計時
      OUT     M32  ; 上燈 1  安定器  異常
      MPP
      OUT     T32 K50  ; 上燈 1  安定器  異常計時
1271  LD      X1D  ; 上燈 1  安定器 Ready
      AND     M397  ; 上燈 1  點燈選擇KP
      AND     M671  ; 點燈時間到達
      LD      M33  ; 上燈 1  點燈失敗
      ANI     M140  ; 警報復歸
      ORB
      MPS
      AND     T33  ; 上燈 1  點燈失敗計時
      OUT     M33  ; 上燈 1  點燈失敗
      MPP
      OUT     T33 K30  ; 上燈 1  點燈失敗計時
1285  LDI     X1E  ; 上燈 2  安定器異常
      LD      M34  ; 上燈 2  安定器  異常
      ANI     M140  ; 警報復歸
      ORB
      MPS
      AND     T34  ; 上燈 2  安定器  異常計時
      OUT     M34  ; 上燈 2  安定器  異常
      MPP
      OUT     T34 K50  ; 上燈 2  安定器  異常計時
1297  LD      X1F  ; 上燈 2  安定器 Ready
      AND     M398  ; 上燈 2  點燈選擇KP
      AND     M671  ; 點燈時間到達
      LD      M35  ; 上燈 2  點燈失敗
      ANI     M140  ; 警報復歸
      ORB
      MPS
      AND     T35  ; 上燈 2  點燈失敗計時
      OUT     M35  ; 上燈 2  點燈失敗
      MPP
      OUT     T35 K30  ; 上燈 2  點燈失敗計時
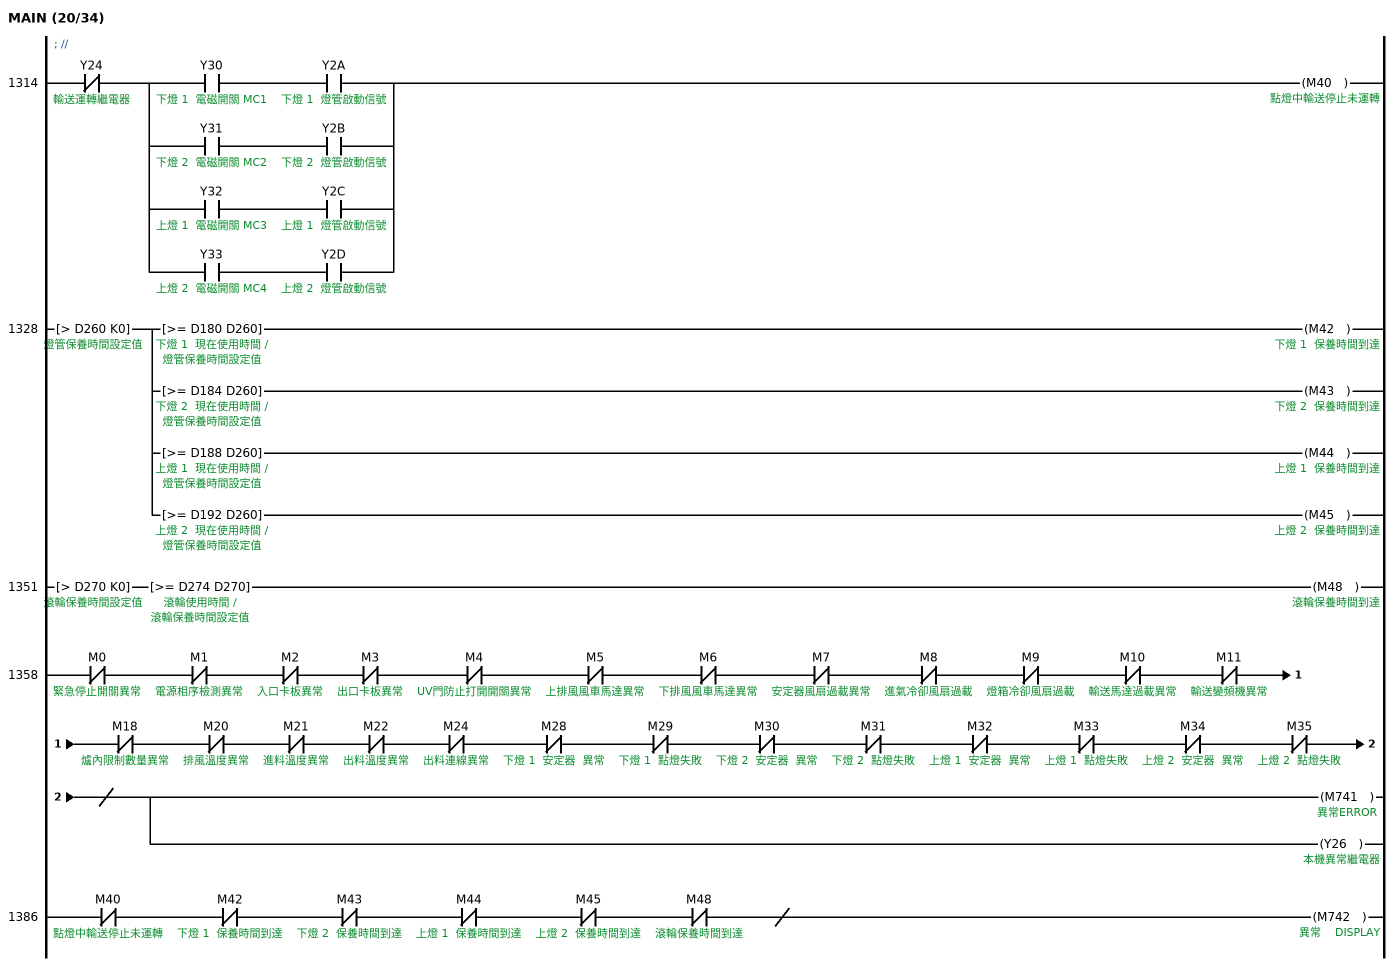
; //
1314  LDI     Y24  ; 輸送運轉繼電器
      LD      Y30  ; 下燈 1  電磁開關 MC1
      AND     Y2A  ; 下燈 1  燈管啟動信號
      LD      Y31  ; 下燈 2  電磁開關 MC2
      AND     Y2B  ; 下燈 2  燈管啟動信號
      ORB
      LD      Y32  ; 上燈 1  電磁開關 MC3
      AND     Y2C  ; 上燈 1  燈管啟動信號
      ORB
      LD      Y33  ; 上燈 2  電磁開關 MC4
      AND     Y2D  ; 上燈 2  燈管啟動信號
      ORB
      ANB
      OUT     M40  ; 點燈中輸送停止未運轉
1328  LD>     D260 K0  ; 燈管保養時間設定值
      MPS
      AND>=   D180 D260  ; 下燈 1  現在使用時間 / 燈管保養時間設定值
      OUT     M42  ; 下燈 1  保養時間到達
      MRD
      AND>=   D184 D260  ; 下燈 2  現在使用時間 / 燈管保養時間設定值
      OUT     M43  ; 下燈 2  保養時間到達
      MRD
      AND>=   D188 D260  ; 上燈 1  現在使用時間 / 燈管保養時間設定值
      OUT     M44  ; 上燈 1  保養時間到達
      MPP
      AND>=   D192 D260  ; 上燈 2  現在使用時間 / 燈管保養時間設定值
      OUT     M45  ; 上燈 2  保養時間到達
1351  LD>     D270 K0  ; 滾輪保養時間設定值
      AND>=   D274 D270  ; 滾輪使用時間 / 滾輪保養時間設定值
      OUT     M48  ; 滾輪保養時間到達
1358  LDI     M0  ; 緊急停止開關異常
      ANI     M1  ; 電源相序檢測異常
      ANI     M2  ; 入口卡板異常
      ANI     M3  ; 出口卡板異常
      ANI     M4  ; UV門防止打開開關異常
      ANI     M5  ; 上排風風車馬達異常
      ANI     M6  ; 下排風風車馬達異常
      ANI     M7  ; 安定器風扇過載異常
      ANI     M8  ; 進氣冷卻風扇過載
      ANI     M9  ; 燈箱冷卻風扇過載
      ANI     M10  ; 輸送馬達過載異常
      ANI     M11  ; 輸送變頻機異常
      ANI     M18  ; 爐內限制數量異常
      ANI     M20  ; 排風溫度異常
      ANI     M21  ; 進料溫度異常
      ANI     M22  ; 出料溫度異常
      ANI     M24  ; 出料連線異常
      ANI     M28  ; 下燈 1  安定器  異常
      ANI     M29  ; 下燈 1  點燈失敗
      ANI     M30  ; 下燈 2  安定器  異常
      ANI     M31  ; 下燈 2  點燈失敗
      ANI     M32  ; 上燈 1  安定器  異常
      ANI     M33  ; 上燈 1  點燈失敗
      ANI     M34  ; 上燈 2  安定器  異常
      ANI     M35  ; 上燈 2  點燈失敗
      INV
      OUT     M741  ; 異常ERROR
      OUT     Y26  ; 本機異常繼電器
1386  LDI     M40  ; 點燈中輸送停止未運轉
      ANI     M42  ; 下燈 1  保養時間到達
      ANI     M43  ; 下燈 2  保養時間到達
      ANI     M44  ; 上燈 1  保養時間到達
      ANI     M45  ; 上燈 2  保養時間到達
      ANI     M48  ; 滾輪保養時間到達
      INV
      OUT     M742  ; 異常    DISPLAY
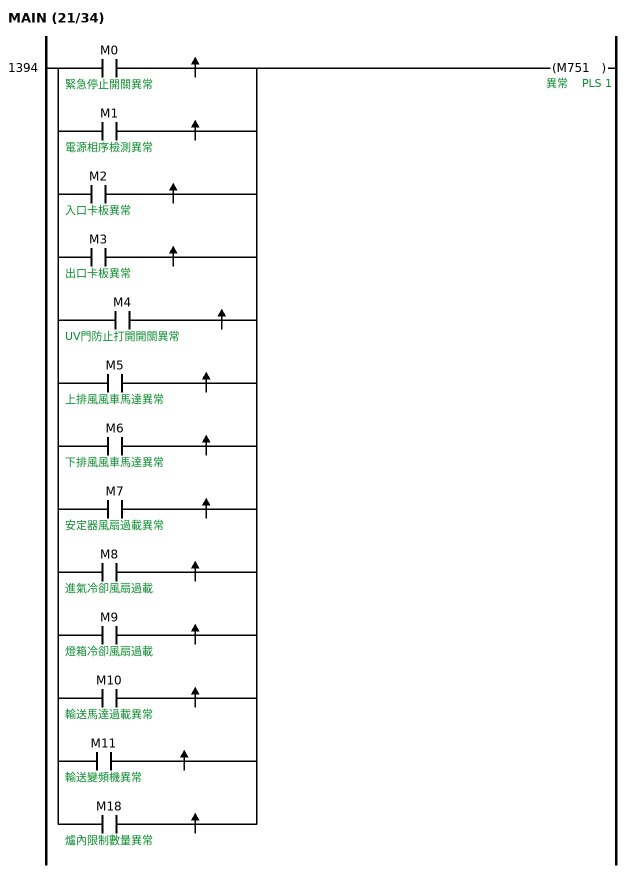
1394  LD      M0  ; 緊急停止開關異常
      MEP
      LD      M1  ; 電源相序檢測異常
      MEP
      ORB
      LD      M2  ; 入口卡板異常
      MEP
      ORB
      LD      M3  ; 出口卡板異常
      MEP
      ORB
      LD      M4  ; UV門防止打開開關異常
      MEP
      ORB
      LD      M5  ; 上排風風車馬達異常
      MEP
      ORB
      LD      M6  ; 下排風風車馬達異常
      MEP
      ORB
      LD      M7  ; 安定器風扇過載異常
      MEP
      ORB
      LD      M8  ; 進氣冷卻風扇過載
      MEP
      ORB
      LD      M9  ; 燈箱冷卻風扇過載
      MEP
      ORB
      LD      M10  ; 輸送馬達過載異常
      MEP
      ORB
      LD      M11  ; 輸送變頻機異常
      MEP
      ORB
      LD      M18  ; 爐內限制數量異常
      MEP
      ORB
      OUT     M751  ; 異常    PLS 1
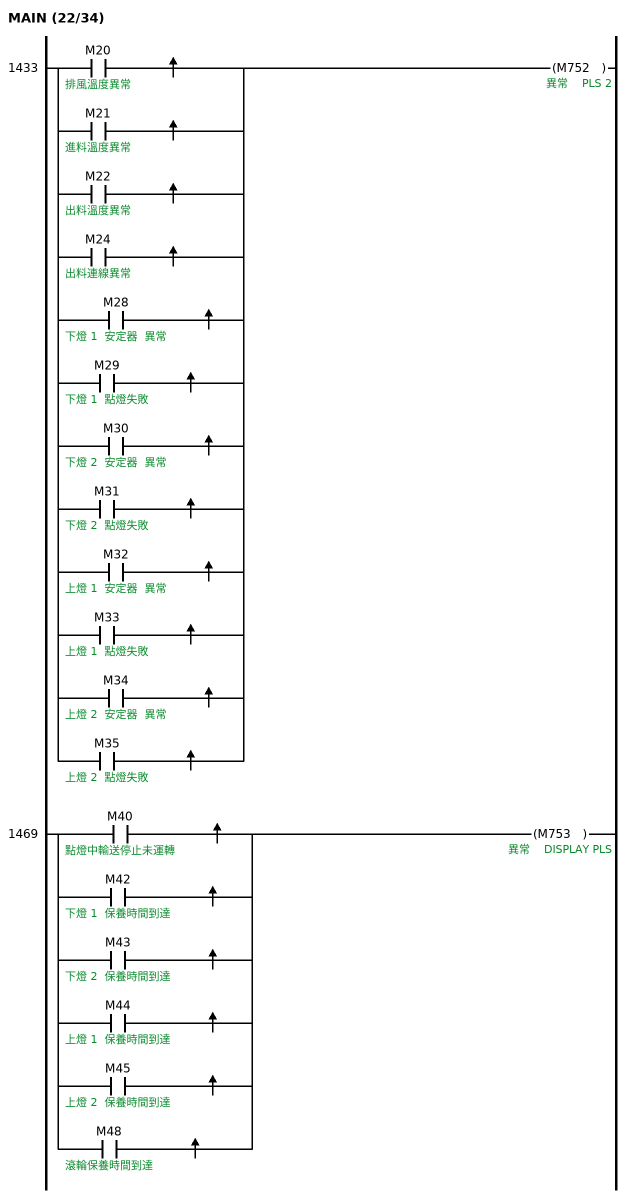
1433  LD      M20  ; 排風溫度異常
      MEP
      LD      M21  ; 進料溫度異常
      MEP
      ORB
      LD      M22  ; 出料溫度異常
      MEP
      ORB
      LD      M24  ; 出料連線異常
      MEP
      ORB
      LD      M28  ; 下燈 1  安定器  異常
      MEP
      ORB
      LD      M29  ; 下燈 1  點燈失敗
      MEP
      ORB
      LD      M30  ; 下燈 2  安定器  異常
      MEP
      ORB
      LD      M31  ; 下燈 2  點燈失敗
      MEP
      ORB
      LD      M32  ; 上燈 1  安定器  異常
      MEP
      ORB
      LD      M33  ; 上燈 1  點燈失敗
      MEP
      ORB
      LD      M34  ; 上燈 2  安定器  異常
      MEP
      ORB
      LD      M35  ; 上燈 2  點燈失敗
      MEP
      ORB
      OUT     M752  ; 異常    PLS 2
1469  LD      M40  ; 點燈中輸送停止未運轉
      MEP
      LD      M42  ; 下燈 1  保養時間到達
      MEP
      ORB
      LD      M43  ; 下燈 2  保養時間到達
      MEP
      ORB
      LD      M44  ; 上燈 1  保養時間到達
      MEP
      ORB
      LD      M45  ; 上燈 2  保養時間到達
      MEP
      ORB
      LD      M48  ; 滾輪保養時間到達
      MEP
      ORB
      OUT     M753  ; 異常    DISPLAY PLS
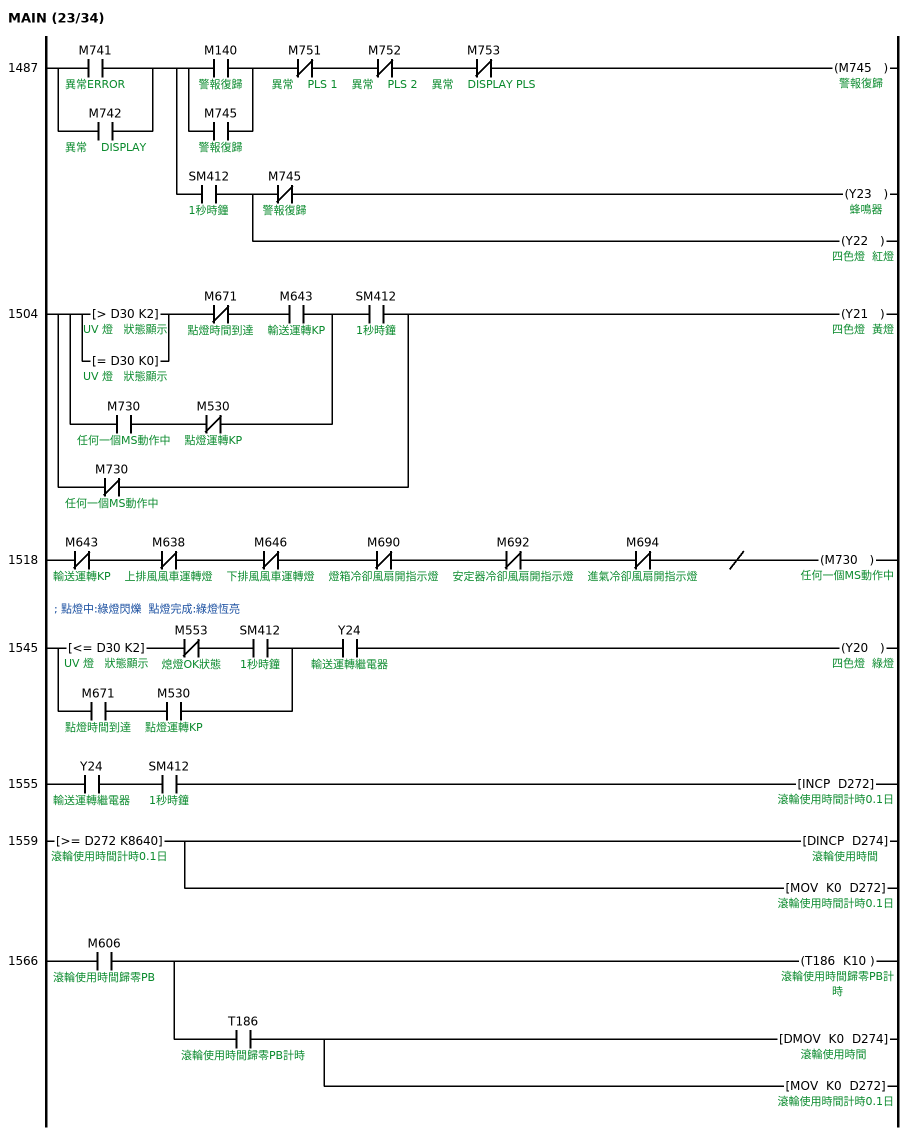
1487  LD      M741  ; 異常ERROR
      OR      M742  ; 異常    DISPLAY
      MPS
      LD      M140  ; 警報復歸
      OR      M745  ; 警報復歸
      ANB
      ANI     M751  ; 異常    PLS 1
      ANI     M752  ; 異常    PLS 2
      ANI     M753  ; 異常    DISPLAY PLS
      OUT     M745  ; 警報復歸
      MPP
      AND     SM412  ; 1秒時鐘
      MPS
      ANI     M745  ; 警報復歸
      OUT     Y23  ; 蜂鳴器
      MPP
      OUT     Y22  ; 四色燈  紅燈
1504  LD>     D30 K2  ; UV 燈   狀態顯示
      OR=     D30 K0  ; UV 燈   狀態顯示
      ANI     M671  ; 點燈時間到達
      AND     M643  ; 輸送運轉KP
      LD      M730  ; 任何一個MS動作中
      ANI     M530  ; 點燈運轉KP
      ORB
      AND     SM412  ; 1秒時鐘
      ORI     M730  ; 任何一個MS動作中
      OUT     Y21  ; 四色燈  黃燈
1518  LDI     M643  ; 輸送運轉KP
      ANI     M638  ; 上排風風車運轉燈
      ANI     M646  ; 下排風風車運轉燈
      ANI     M690  ; 燈箱冷卻風扇開指示燈
      ANI     M692  ; 安定器冷卻風扇開指示燈
      ANI     M694  ; 進氣冷卻風扇開指示燈
      INV
      OUT     M730  ; 任何一個MS動作中
; 點燈中:綠燈閃爍  點燈完成:綠燈恆亮
1545  LD<=    D30 K2  ; UV 燈   狀態顯示
      ANI     M553  ; 熄燈OK狀態
      AND     SM412  ; 1秒時鐘
      LD      M671  ; 點燈時間到達
      AND     M530  ; 點燈運轉KP
      ORB
      AND     Y24  ; 輸送運轉繼電器
      OUT     Y20  ; 四色燈  綠燈
1555  LD      Y24  ; 輸送運轉繼電器
      AND     SM412  ; 1秒時鐘
      INCP    D272  ; 滾輪使用時間計時0.1日
1559  LD>=    D272 K8640  ; 滾輪使用時間計時0.1日
      DINCP   D274
      MOV     K0 D272
1566  LD      M606  ; 滾輪使用時間歸零PB
      OUT     T186 K10  ; 滾輪使用時間歸零PB計時
      AND     T186  ; 滾輪使用時間歸零PB計時
      DMOV    K0 D274
      MOV     K0 D272
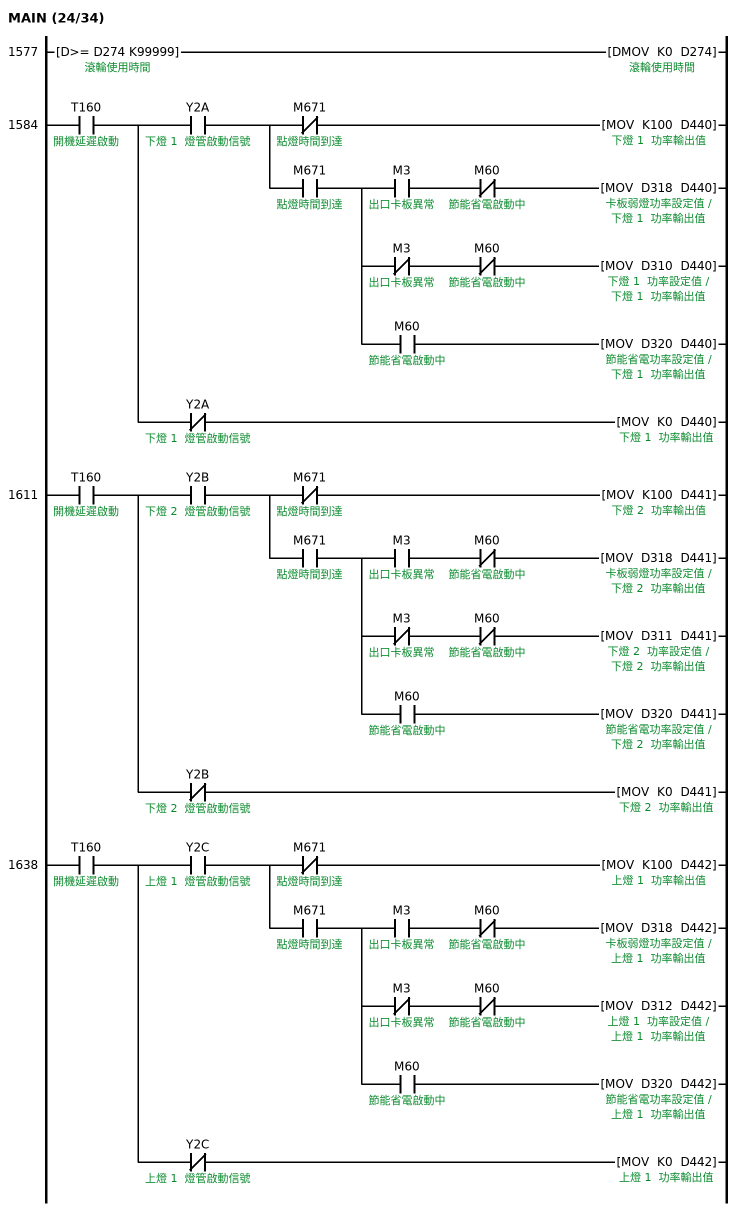
1577  LDD>=   D274 K99999  ; 滾輪使用時間
      DMOV    K0 D274
1584  LD      T160  ; 開機延遲啟動
      MPS
      AND     Y2A  ; 下燈 1  燈管啟動信號
      MPS
      ANI     M671  ; 點燈時間到達
      MOV     K100 D440  ; 下燈 1  功率輸出值
      MPP
      AND     M671  ; 點燈時間到達
      MPS
      AND     M3  ; 出口卡板異常
      ANI     M60  ; 節能省電啟動中
      MOV     D318 D440
      MRD
      ANI     M3  ; 出口卡板異常
      ANI     M60  ; 節能省電啟動中
      MOV     D310 D440
      MPP
      AND     M60  ; 節能省電啟動中
      MOV     D320 D440
      MPP
      ANI     Y2A  ; 下燈 1  燈管啟動信號
      MOV     K0 D440
1611  LD      T160  ; 開機延遲啟動
      MPS
      AND     Y2B  ; 下燈 2  燈管啟動信號
      MPS
      ANI     M671  ; 點燈時間到達
      MOV     K100 D441  ; 下燈 2  功率輸出值
      MPP
      AND     M671  ; 點燈時間到達
      MPS
      AND     M3  ; 出口卡板異常
      ANI     M60  ; 節能省電啟動中
      MOV     D318 D441
      MRD
      ANI     M3  ; 出口卡板異常
      ANI     M60  ; 節能省電啟動中
      MOV     D311 D441
      MPP
      AND     M60  ; 節能省電啟動中
      MOV     D320 D441
      MPP
      ANI     Y2B  ; 下燈 2  燈管啟動信號
      MOV     K0 D441
1638  LD      T160  ; 開機延遲啟動
      MPS
      AND     Y2C  ; 上燈 1  燈管啟動信號
      MPS
      ANI     M671  ; 點燈時間到達
      MOV     K100 D442  ; 上燈 1  功率輸出值
      MPP
      AND     M671  ; 點燈時間到達
      MPS
      AND     M3  ; 出口卡板異常
      ANI     M60  ; 節能省電啟動中
      MOV     D318 D442
      MRD
      ANI     M3  ; 出口卡板異常
      ANI     M60  ; 節能省電啟動中
      MOV     D312 D442
      MPP
      AND     M60  ; 節能省電啟動中
      MOV     D320 D442
      MPP
      ANI     Y2C  ; 上燈 1  燈管啟動信號
      MOV     K0 D442
